KUKA KRL program: EPS_2_251349_MH89A_A_20250929014701.src

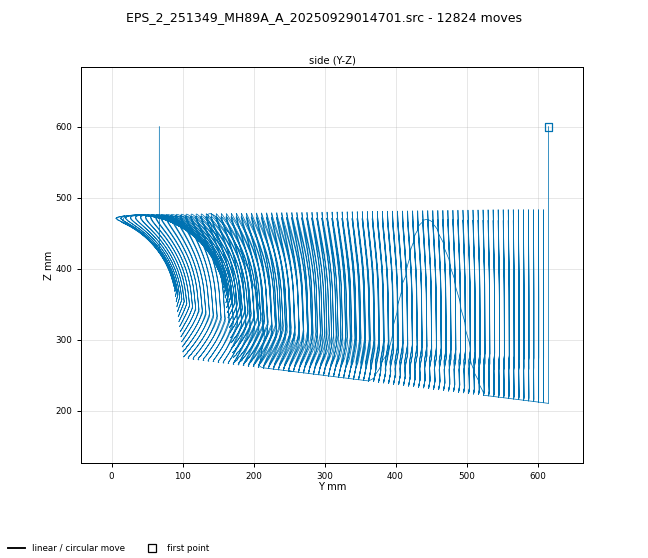
[picture p0: tool path of EPS_2_251349_MH89A_A_20250929014701.src, 12824 of 12826 moves have a stored position in this frame; points joined in program order, loops and branches not executed]
&ACCESS RVP
&REL 4
&COMMENT QRS 19112012
&PARAM EDITMASK = *
DEF PART()
EXT BAS (BAS_COMMAND :IN,REAL :IN )
INT I
BAS (#INITMOV,0 )

;KUKA QRS Post kuka4.cps  Date:22-06-2017 !

File_ID=2864

QRS_PRE_INIT()

;Init var - Until changes are made in qrs_pre_init
Outlet_Square_prg=0
Inlet_1_Square_prg=0
Inlet_2_Square_prg=0
Inlet_3_Square_prg=0
Inlet_4_Square_prg=0
Inlet_5_Square_prg=0

Outlet_1={X 0.000, Y 540.910, Z 382.500, B 0.000, E1 0.000 }
Inlet_1={X 0.000, Y 541.980, Z 367.500, B 0.000, E1 157.000 }
Outlet_1_type=201
Inlet_1_type=201
;QRS#1=Sidecore dimensions
;QRS#2=200-8" PVC SDR 35
;QRS#3=200-8" PVC SDR 35
;QRS#4=
;QRS#5=
;QRS#6=
;QRS#7=
;QRS#8=
;QRS#9=12-08 PSX
;QRS#10=12-08 PSX
;QRS#11=
;QRS#12=
;QRS#13=
;QRS#14=
;QRS#15=
;QRS#16=1220x127x762 2,5'
;QRS#17=EPS Height
;QRS#18=483
;QRS#19=*
;QRS#20= UPDATED VERSION 22-06-2017
;QRS#21=*
Outlet_Square=0100
Inlet_1_Square=0100
Inlet_2_Square=0
Inlet_3_Square=0
Inlet_4_Square=0
Inlet_5_Square=0
Mill_Square=1
Outlet_Square_Prg=204
Inlet_1_Square_prg=204

QRS_INIT()

$ADVANCE=5

; T1
PTP {E1 173.665,E2 173.665}
PTP {X 0,Y 615.418,A -85,B 0,C 180,E1 173.665,E2 173.665,E3 0,E4 0,E5 0,E6 0}
QRS_SPEED_INIT()
LIN {X 0,Y 615.418,Z 600,A -85,B 0,C 180,E1 173.665,E2 173.665,E3 0,E4 0,E5 0,E6 0} C_VEL
LIN {X 0,Y 615.418,Z 220.378,A -85,B 0,C 180,E1 173.665,E2 173.665} C_VEL
LIN {X 0,Y 615.418,Z 212.2,A -85,B 0,C 180,E1 173.665,E2 173.665} C_VEL
LIN {X 0,Y 615.407,Z 210.2,A -85,B 0,C 180,E1 173.479,E2 173.479} C_VEL
LIN {X 0,Y 615.411,Z 210.199,A -85,B 0,C 180,E1 171.465,E2 171.465} C_VEL
LIN {X 0,Y 615.419,Z 210.199,A -85,B 0,C 180,E1 169.475,E2 169.475} C_VEL
LIN {X 0,Y 615.425,Z 210.198,A -85,B 0,C 180,E1 167.471,E2 167.471} C_VEL
LIN {X 0,Y 615.431,Z 210.197,A -85,B 0,C 180,E1 165.452,E2 165.452} C_VEL
LIN {X 0,Y 615.437,Z 210.196,A -85,B 0,C 180,E1 163.415,E2 163.415} C_VEL
LIN {X 0,Y 615.44,Z 210.196,A -85,B 0,C 180,E1 161.356,E2 161.356} C_VEL
LIN {X 0,Y 615.441,Z 210.195,A -85,B 0,C 180,E1 159.271,E2 159.271} C_VEL
LIN {X 0,Y 615.438,Z 210.195,A -85,B 0,C 180,E1 157.157,E2 157.157} C_VEL
LIN {X 0,Y 615.434,Z 210.194,A -85,B 0,C 180,E1 155.009,E2 155.009} C_VEL
LIN {X 0,Y 615.429,Z 210.194,A -85,B 0,C 180,E1 152.824,E2 152.824} C_VEL
LIN {X 0,Y 615.425,Z 210.195,A -85,B 0,C 180,E1 150.594,E2 150.594} C_VEL
LIN {X 0,Y 615.425,Z 210.196,A -85,B 0,C 180,E1 148.315,E2 148.315} C_VEL
LIN {X 0,Y 615.44,Z 210.197,A -85,B 0,C 180,E1 145.979,E2 145.979} C_VEL
LIN {X 0,Y 615.468,Z 210.2,A -85,B 0,C 180,E1 143.578,E2 143.578} C_VEL
LIN {X 0,Y 615.489,Z 210.188,A -85,B 0,C 180,E1 140.936,E2 140.936} C_VEL
LIN {X 0,Y 615.454,Z 210.19,A -85,B 0,C 180,E1 138.528,E2 138.528} C_VEL
LIN {X 0,Y 615.437,Z 210.193,A -85,B 0,C 180,E1 136.006,E2 136.006} C_VEL
LIN {X 0,Y 615.439,Z 210.192,A -85,B 0,C 180,E1 133.998,E2 133.998} C_VEL
LIN {X 0,Y 615.491,Z 210.391,A -85,B 0,C 180,E1 133.031,E2 133.031} C_VEL
LIN {X 0,Y 615.494,Z 227.3,A -85,B 0,C 180,E1 130.35,E2 130.35} C_VEL
LIN {X 0,Y 615.432,Z 244.862,A -85,B 0,C 180,E1 127.63,E2 127.63} C_VEL
LIN {X 0,Y 615.441,Z 256.667,A -85,B 0,C 180,E1 125.853,E2 125.853} C_VEL
LIN {X 0,Y 615.439,Z 257.703,A -85,B 0,C 180,E1 125.807,E2 125.807} C_VEL
LIN {X 0,Y 615.498,Z 364.309,A -85,B 0,C 180,E1 124.535,E2 124.535} C_VEL
LIN {X 0,Y 615.496,Z 377.737,A -85,B 0,C 180,E1 124.235,E2 124.235} C_VEL
LIN {X 0,Y 615.497,Z 389.639,A -85,B 0,C 180,E1 123.841,E2 123.841} C_VEL
LIN {X 0,Y 615.48,Z 401.538,A -85,B 0,C 180,E1 123.313,E2 123.313} C_VEL
LIN {X 0,Y 615.477,Z 412.999,A -85,B 0,C 180,E1 122.651,E2 122.651} C_VEL
LIN {X 0,Y 615.498,Z 424.079,A -85,B 0,C 180,E1 121.847,E2 121.847} C_VEL
LIN {X 0,Y 615.495,Z 432.368,A -85,B 0,C 180,E1 121.095,E2 121.095} C_VEL
LIN {X 0,Y 615.493,Z 439.497,A -85,B 0,C 180,E1 120.348,E2 120.348} C_VEL
LIN {X 0,Y 615.487,Z 446.811,A -85,B 0,C 180,E1 119.405,E2 119.405} C_VEL
LIN {X 0,Y 615.496,Z 452.759,A -85,B 0,C 180,E1 118.46,E2 118.46} C_VEL
LIN {X 0,Y 615.495,Z 457.422,A -85,B 0,C 180,E1 117.544,E2 117.544} C_VEL
LIN {X 0,Y 615.496,Z 461.71,A -85,B 0,C 180,E1 116.443,E2 116.443} C_VEL
LIN {X 0,Y 615.494,Z 464.217,A -85,B 0,C 180,E1 115.579,E2 115.579} C_VEL
LIN {X 0,Y 615.498,Z 465.487,A -85,B 0,C 180,E1 114.99,E2 114.99} C_VEL
LIN {X 0,Y 615.495,Z 466.868,A -85,B 0,C 180,E1 114.02,E2 114.02} C_VEL
LIN {X 0,Y 615.492,Z 467.368,A -85,B 0,C 180,E1 112.844,E2 112.844} C_VEL
LIN {X 0,Y 615.497,Z 467.056,A -85,B 0,C 180,E1 112.135,E2 112.135} C_VEL
LIN {X 0,Y 615.496,Z 466.325,A -85,B 0,C 180,E1 111.431,E2 111.431} C_VEL
LIN {X 0,Y 615.496,Z 464.751,A -85,B 0,C 180,E1 110.571,E2 110.571} C_VEL
LIN {X 0,Y 615.497,Z 461.291,A -85,B 0,C 180,E1 109.337,E2 109.337} C_VEL
LIN {X 0,Y 615.496,Z 457.068,A -85,B 0,C 180,E1 108.287,E2 108.287} C_VEL
LIN {X 0,Y 615.497,Z 450.678,A -85,B 0,C 180,E1 107.098,E2 107.098} C_VEL
LIN {X 0,Y 615.498,Z 443.391,A -85,B 0,C 180,E1 106.04,E2 106.04} C_VEL
LIN {X 0,Y 615.497,Z 436.479,A -85,B 0,C 180,E1 105.225,E2 105.225} C_VEL
LIN {X 0,Y 615.498,Z 426.304,A -85,B 0,C 180,E1 104.251,E2 104.251} C_VEL
LIN {X 0,Y 615.492,Z 415.94,A -85,B 0,C 180,E1 103.453,E2 103.453} C_VEL
LIN {X 0,Y 615.47,Z 405,A -85,B 0,C 180,E1 102.781,E2 102.781} C_VEL
LIN {X 0,Y 615.498,Z 392.743,A -85,B 0,C 180,E1 102.194,E2 102.194} C_VEL
LIN {X 0,Y 615.498,Z 379.878,A -85,B 0,C 180,E1 101.735,E2 101.735} C_VEL
LIN {X 0,Y 615.498,Z 366.871,A -85,B 0,C 180,E1 101.422,E2 101.422} C_VEL
LIN {X 0,Y 615.496,Z 348.647,A -85,B 0,C 180,E1 101.174,E2 101.174} C_VEL
LIN {X 0,Y 615.43,Z 257.274,A -85,B 0,C 180,E1 100.091,E2 100.091} C_VEL
LIN {X 0,Y 615.432,Z 256.35,A -85,B 0,C 180,E1 100.029,E2 100.029} C_VEL
LIN {X 0,Y 615.495,Z 239.011,A -85,B 0,C 180,E1 97.38,E2 97.38} C_VEL
LIN {X 0,Y 615.47,Z 221.075,A -85,B 0,C 180,E1 94.584,E2 94.584} C_VEL
LIN {X 0,Y 615.498,Z 210.337,A -85,B 0,C 180,E1 92.863,E2 92.863} C_VEL
LIN {X 0,Y 615.484,Z 210.201,A -85,B 0,C 180,E1 90.654,E2 90.654} C_VEL
LIN {X 0,Y 615.432,Z 210.196,A -85,B 0,C 180,E1 88.036,E2 88.036} C_VEL
LIN {X 0,Y 615.437,Z 210.197,A -85,B 0,C 180,E1 86.071,E2 86.071} C_VEL
LIN {X 0,Y 615.445,Z 210.198,A -85,B 0,C 180,E1 84.101,E2 84.101} C_VEL
LIN {X 0,Y 615.453,Z 210.198,A -85,B 0,C 180,E1 82.123,E2 82.123} C_VEL
LIN {X 0,Y 615.462,Z 210.199,A -85,B 0,C 180,E1 80.137,E2 80.137} C_VEL
LIN {X 0,Y 615.419,Z 210.197,A -85,B 0,C 180,E1 77.468,E2 77.468} C_VEL
LIN {X 0,Y 615.42,Z 210.197,A -85,B 0,C 180,E1 75.449,E2 75.449} C_VEL
LIN {X 0,Y 615.419,Z 210.197,A -85,B 0,C 180,E1 73.411,E2 73.411} C_VEL
LIN {X 0,Y 615.419,Z 210.197,A -85,B 0,C 180,E1 71.351,E2 71.351} C_VEL
LIN {X 0,Y 615.417,Z 210.198,A -85,B 0,C 180,E1 69.266,E2 69.266} C_VEL
LIN {X 0,Y 615.415,Z 210.198,A -85,B 0,C 180,E1 67.152,E2 67.152} C_VEL
LIN {X 0,Y 615.412,Z 210.198,A -85,B 0,C 180,E1 65.005,E2 65.005} C_VEL
LIN {X 0,Y 615.411,Z 210.198,A -85,B 0,C 180,E1 62.819,E2 62.819} C_VEL
LIN {X 0,Y 615.444,Z 210.197,A -85,B 0,C 180,E1 60.205,E2 60.205} C_VEL
LIN {X 0,Y 615.478,Z 210.2,A -85,B 0,C 180,E1 57.542,E2 57.542} C_VEL
LIN {X 0,Y 615.438,Z 210.2,A -85,B 0,C 180,E1 55.181,E2 55.181} C_VEL
LIN {X 0,Y 615.409,Z 210.199,A -85,B 0,C 180,E1 52.752,E2 52.752} C_VEL
LIN {X 0,Y 615.406,Z 210.2,A -85,B 0,C 180,E1 50.243,E2 50.243} C_VEL
LIN {X 0,Y 615.451,Z 210.2,A -85,B 0,C 180,E1 47.644,E2 47.644} C_VEL
LIN {X 0,Y 615.447,Z 210.2,A -85,B 0,C 180,E1 44.927,E2 44.927} C_VEL
LIN {X 0,Y 615.471,Z 210.2,A -85,B 0,C 180,E1 43.045,E2 43.045} C_VEL
LIN {X 0,Y 615.43,Z 210.199,A -85,B 0,C 180,E1 40.606,E2 40.606} C_VEL
LIN {X 0,Y 615.48,Z 210.198,A -85,B 0,C 180,E1 38.9,E2 38.9} C_VEL
LIN {X 0,Y 615.43,Z 210.198,A -85,B 0,C 180,E1 36.425,E2 36.425} C_VEL
LIN {X 0,Y 615.411,Z 210.198,A -85,B 0,C 180,E1 34.023,E2 34.023} C_VEL
LIN {X 0,Y 615.411,Z 210.198,A -85,B 0,C 180,E1 31.686,E2 31.686} C_VEL
LIN {X 0,Y 615.42,Z 210.198,A -85,B 0,C 180,E1 29.406,E2 29.406} C_VEL
LIN {X 0,Y 615.447,Z 210.199,A -85,B 0,C 180,E1 27.037,E2 27.037} C_VEL
LIN {X 0,Y 615.439,Z 210.195,A -85,B 0,C 180,E1 23.998,E2 23.998} C_VEL
LIN {X 0,Y 615.463,Z 210.194,A -85,B 0,C 180,E1 22.134,E2 22.134} C_VEL
LIN {X 0,Y 615.461,Z 210.194,A -85,B 0,C 180,E1 20.031,E2 20.031} C_VEL
LIN {X 0,Y 615.462,Z 210.193,A -85,B 0,C 180,E1 17.955,E2 17.955} C_VEL
LIN {X 0,Y 615.466,Z 210.193,A -85,B 0,C 180,E1 15.903,E2 15.903} C_VEL
LIN {X 0,Y 615.422,Z 210.195,A -85,B 0,C 180,E1 13.2,E2 13.2} C_VEL
LIN {X 0,Y 615.424,Z 210.197,A -85,B 0,C 180,E1 10.857,E2 10.857} C_VEL
LIN {X 0,Y 615.442,Z 210.198,A -85,B 0,C 180,E1 8.535,E2 8.535} C_VEL
LIN {X 0,Y 615.497,Z 210.196,A -85,B 0,C 180,E1 5.896,E2 5.896} C_VEL
LIN {X 0,Y 615.452,Z 210.191,A -85,B 0,C 180,E1 3.271,E2 3.271} C_VEL
LIN {X 0,Y 615.465,Z 210.19,A -85,B 0,C 180,E1 1.306,E2 1.306} C_VEL
LIN {X 0,Y 615.43,Z 210.194,A -85,B 0,C 180,E1 -1.311,E2 -1.311} C_VEL
LIN {X 0,Y 615.434,Z 210.192,A -85,B 0,C 180,E1 -3.275,E2 -3.275} C_VEL
LIN {X 0,Y 615.439,Z 210.192,A -85,B 0,C 180,E1 -5.244,E2 -5.244} C_VEL
LIN {X 0,Y 615.448,Z 210.19,A -85,B 0,C 180,E1 -7.218,E2 -7.218} C_VEL
LIN {X 0,Y 615.456,Z 210.189,A -85,B 0,C 180,E1 -9.201,E2 -9.201} C_VEL
LIN {X 0,Y 615.465,Z 210.188,A -85,B 0,C 180,E1 -11.195,E2 -11.195} C_VEL
LIN {X 0,Y 615.472,Z 210.188,A -85,B 0,C 180,E1 -13.203,E2 -13.203} C_VEL
LIN {X 0,Y 615.438,Z 210.193,A -85,B 0,C 180,E1 -15.908,E2 -15.908} C_VEL
LIN {X 0,Y 615.473,Z 210.199,A -85,B 0,C 180,E1 -18.6,E2 -18.6} C_VEL
LIN {X 0,Y 615.484,Z 210.185,A -85,B 0,C 180,E1 -21.434,E2 -21.434} C_VEL
LIN {X 0,Y 615.445,Z 210.19,A -85,B 0,C 180,E1 -23.999,E2 -23.999} C_VEL
LIN {X 0,Y 615.444,Z 210.194,A -85,B 0,C 180,E1 -26.448,E2 -26.448} C_VEL
LIN {X 0,Y 615.493,Z 210.191,A -85,B 0,C 180,E1 -29.407,E2 -29.407} C_VEL
LIN {X 0,Y 615.489,Z 210.186,A -85,B 0,C 180,E1 -31.687,E2 -31.687} C_VEL
LIN {X 0,Y 615.473,Z 210.185,A -85,B 0,C 180,E1 -34.024,E2 -34.024} C_VEL
LIN {X 0,Y 615.451,Z 210.189,A -85,B 0,C 180,E1 -36.429,E2 -36.429} C_VEL
LIN {X 0,Y 615.46,Z 210.195,A -85,B 0,C 180,E1 -39.059,E2 -39.059} C_VEL
LIN {X 0,Y 615.49,Z 210.201,A -85,B 0,C 180,E1 -41.475,E2 -41.475} C_VEL
LIN {X 0,Y 615.496,Z 210.183,A -85,B 0,C 180,E1 -44.15,E2 -44.15} C_VEL
LIN {X 0,Y 615.453,Z 210.19,A -85,B 0,C 180,E1 -46.957,E2 -46.957} C_VEL
LIN {X 0,Y 615.463,Z 210.195,A -85,B 0,C 180,E1 -49.391,E2 -49.391} C_VEL
LIN {X 0,Y 615.493,Z 210.196,A -85,B 0,C 180,E1 -51.989,E2 -51.989} C_VEL
LIN {X 0,Y 615.49,Z 210.187,A -85,B 0,C 180,E1 -54.384,E2 -54.384} C_VEL
LIN {X 0,Y 615.486,Z 210.182,A -85,B 0,C 180,E1 -56.763,E2 -56.763} C_VEL
LIN {X 0,Y 615.472,Z 210.184,A -85,B 0,C 180,E1 -59.079,E2 -59.079} C_VEL
LIN {X 0,Y 615.46,Z 210.19,A -85,B 0,C 180,E1 -61.556,E2 -61.556} C_VEL
LIN {X 0,Y 615.498,Z 210.199,A -85,B 0,C 180,E1 -64.284,E2 -64.284} C_VEL
LIN {X 0,Y 615.484,Z 210.182,A -85,B 0,C 180,E1 -67.155,E2 -67.155} C_VEL
LIN {X 0,Y 615.492,Z 210.437,A -85,B 0,C 180,E1 -68.48,E2 -68.48} C_VEL
LIN {X 0,Y 615.494,Z 228.957,A -85,B 0,C 180,E1 -71.181,E2 -71.181} C_VEL
LIN {X 0,Y 615.488,Z 249.421,A -85,B 0,C 180,E1 -74.094,E2 -74.094} C_VEL
LIN {X 0,Y 615.473,Z 268.661,A -85,B 0,C 180,E1 -76.798,E2 -76.798} C_VEL
LIN {X 0,Y 615.487,Z 271.24,A -85,B 0,C 180,E1 -77.113,E2 -77.113} C_VEL
LIN {X 0,Y 615.491,Z 280.005,A -85,B 0,C 180,E1 -77.239,E2 -77.239} C_VEL
LIN {X 0,Y 615.498,Z 378.802,A -85,B 0,C 180,E1 -78.41,E2 -78.41} C_VEL
LIN {X 0,Y 615.498,Z 391.325,A -85,B 0,C 180,E1 -78.682,E2 -78.682} C_VEL
LIN {X 0,Y 615.496,Z 404.513,A -85,B 0,C 180,E1 -79.109,E2 -79.109} C_VEL
LIN {X 0,Y 615.491,Z 416.467,A -85,B 0,C 180,E1 -79.639,E2 -79.639} C_VEL
LIN {X 0,Y 615.48,Z 427.989,A -85,B 0,C 180,E1 -80.303,E2 -80.303} C_VEL
LIN {X 0,Y 615.499,Z 438.335,A -85,B 0,C 180,E1 -81.049,E2 -81.049} C_VEL
LIN {X 0,Y 615.498,Z 446.687,A -85,B 0,C 180,E1 -81.794,E2 -81.794} C_VEL
LIN {X 0,Y 615.498,Z 454.602,A -85,B 0,C 180,E1 -82.619,E2 -82.619} C_VEL
LIN {X 0,Y 615.49,Z 462.201,A -85,B 0,C 180,E1 -83.607,E2 -83.607} C_VEL
LIN {X 0,Y 615.498,Z 469.202,A -85,B 0,C 180,E1 -84.758,E2 -84.758} C_VEL
LIN {X 0,Y 615.493,Z 473.849,A -85,B 0,C 180,E1 -85.743,E2 -85.743} C_VEL
LIN {X 0,Y 615.494,Z 477.397,A -85,B 0,C 180,E1 -86.727,E2 -86.727} C_VEL
LIN {X 0,Y 615.497,Z 479.232,A -85,B 0,C 180,E1 -87.382,E2 -87.382} C_VEL
LIN {X 0,Y 615.497,Z 480.607,A -85,B 0,C 180,E1 -88.036,E2 -88.036} C_VEL
LIN {X 0,Y 615.496,Z 482.173,A -85,B 0,C 180,E1 -89.345,E2 -89.345} C_VEL
LIN {X 0,Y 615.494,Z 482.389,A -85,B 0,C 180,E1 -89.999,E2 -89.999} C_VEL
LIN {X 0,Y 615.495,Z 481.581,A -85,B 0,C 180,E1 -91.308,E2 -91.308} C_VEL
LIN {X 0,Y 615.497,Z 480.609,A -85,B 0,C 180,E1 -91.963,E2 -91.963} C_VEL
LIN {X 0,Y 615.497,Z 479.234,A -85,B 0,C 180,E1 -92.617,E2 -92.617} C_VEL
LIN {X 0,Y 615.496,Z 476.351,A -85,B 0,C 180,E1 -93.6,E2 -93.6} C_VEL
LIN {X 0,Y 615.498,Z 472.444,A -85,B 0,C 180,E1 -94.584,E2 -94.584} C_VEL
LIN {X 0,Y 615.499,Z 467.408,A -85,B 0,C 180,E1 -95.569,E2 -95.569} C_VEL
LIN {X 0,Y 615.489,Z 460.918,A -85,B 0,C 180,E1 -96.577,E2 -96.577} C_VEL
LIN {X 0,Y 615.497,Z 453.138,A -85,B 0,C 180,E1 -97.545,E2 -97.545} C_VEL
LIN {X 0,Y 615.498,Z 443.264,A -85,B 0,C 180,E1 -98.536,E2 -98.536} C_VEL
LIN {X 0,Y 615.495,Z 432.874,A -85,B 0,C 180,E1 -99.364,E2 -99.364} C_VEL
LIN {X 0,Y 615.475,Z 422.588,A -85,B 0,C 180,E1 -100.028,E2 -100.028} C_VEL
LIN {X 0,Y 615.497,Z 411.108,A -85,B 0,C 180,E1 -100.617,E2 -100.617} C_VEL
LIN {X 0,Y 615.499,Z 399.282,A -85,B 0,C 180,E1 -101.079,E2 -101.079} C_VEL
LIN {X 0,Y 615.498,Z 386.267,A -85,B 0,C 180,E1 -101.442,E2 -101.442} C_VEL
LIN {X 0,Y 615.499,Z 372.989,A -85,B 0,C 180,E1 -101.672,E2 -101.672} C_VEL
LIN {X 0,Y 615.488,Z 271.757,A -85,B 0,C 180,E1 -102.865,E2 -102.865} C_VEL
LIN {X 0,Y 615.485,Z 270.524,A -85,B 0,C 180,E1 -102.949,E2 -102.949} C_VEL
LIN {X 0,Y 615.481,Z 250.632,A -85,B 0,C 180,E1 -105.735,E2 -105.735} C_VEL
LIN {X 0,Y 615.491,Z 231.586,A -85,B 0,C 180,E1 -108.442,E2 -108.442} C_VEL
LIN {X 0,Y 615.492,Z 212.096,A -85,B 0,C 180,E1 -111.255,E2 -111.255} C_VEL
LIN {X 0,Y 615.49,Z 210.315,A -85,B 0,C 180,E1 -111.563,E2 -111.563} C_VEL
LIN {X 0,Y 615.461,Z 210.19,A -85,B 0,C 180,E1 -114.272,E2 -114.272} C_VEL
LIN {X 0,Y 615.497,Z 210.18,A -85,B 0,C 180,E1 -117.046,E2 -117.046} C_VEL
LIN {X 0,Y 615.497,Z 210.199,A -85,B 0,C 180,E1 -119.795,E2 -119.795} C_VEL
LIN {X 0,Y 615.457,Z 210.192,A -85,B 0,C 180,E1 -122.458,E2 -122.458} C_VEL
LIN {X 0,Y 615.456,Z 210.188,A -85,B 0,C 180,E1 -124.816,E2 -124.816} C_VEL
LIN {X 0,Y 615.476,Z 210.184,A -85,B 0,C 180,E1 -127.242,E2 -127.242} C_VEL
LIN {X 0,Y 615.497,Z 210.199,A -85,B 0,C 180,E1 -130.089,E2 -130.089} C_VEL
LIN {X 0,Y 615.481,Z 210.198,A -85,B 0,C 180,E1 -132.352,E2 -132.352} C_VEL
LIN {X 0,Y 615.444,Z 210.191,A -85,B 0,C 180,E1 -135.071,E2 -135.071} C_VEL
LIN {X 0,Y 615.498,Z 210.185,A -85,B 0,C 180,E1 -137.917,E2 -137.917} C_VEL
LIN {X 0,Y 615.495,Z 210.194,A -85,B 0,C 180,E1 -140.249,E2 -140.249} C_VEL
LIN {X 0,Y 615.445,Z 210.195,A -85,B 0,C 180,E1 -143.067,E2 -143.067} C_VEL
LIN {X 0,Y 615.438,Z 210.193,A -85,B 0,C 180,E1 -145.304,E2 -145.304} C_VEL
LIN {X 0,Y 615.441,Z 210.191,A -85,B 0,C 180,E1 -147.674,E2 -147.674} C_VEL
LIN {X 0,Y 615.491,Z 210.197,A -85,B 0,C 180,E1 -150.592,E2 -150.592} C_VEL
LIN {X 0,Y 615.476,Z 210.199,A -85,B 0,C 180,E1 -152.955,E2 -152.955} C_VEL
LIN {X 0,Y 615.476,Z 210.199,A -85,B 0,C 180,E1 -155.006,E2 -155.006} C_VEL
LIN {X 0,Y 615.429,Z 210.195,A -85,B 0,C 180,E1 -157.665,E2 -157.665} C_VEL
LIN {X 0,Y 615.424,Z 210.195,A -85,B 0,C 180,E1 -159.963,E2 -159.963} C_VEL
LIN {X 0,Y 615.481,Z 210.192,A -85,B 0,C 180,E1 -162.728,E2 -162.728} C_VEL
LIN {X 0,Y 615.455,Z 210.199,A -85,B 0,C 180,E1 -165.448,E2 -165.448} C_VEL
LIN {X 0,Y 615.46,Z 210.199,A -85,B 0,C 180,E1 -167.467,E2 -167.467} C_VEL
LIN {X 0,Y 615.463,Z 210.2,A -85,B 0,C 180,E1 -169.471,E2 -169.471} C_VEL
LIN {X 0,Y 615.416,Z 210.198,A -85,B 0,C 180,E1 -172.121,E2 -172.121} C_VEL
LIN {X 0,Y 615.417,Z 210.198,A -85,B 0,C 180,E1 -174.099,E2 -174.099} C_VEL
LIN {X 0,Y 615.419,Z 210.199,A -85,B 0,C 180,E1 -176.069,E2 -176.069} C_VEL
LIN {X 0,Y 615.427,Z 210.199,A -85,B 0,C 180,E1 -178.035,E2 -178.035} C_VEL
LIN {X 0,Y 615.434,Z 210.2,A -85,B 0,C 180,E1 -179.998,E2 -179.998} C_VEL
LIN {X 0,Y 615.444,Z 210.2,A -85,B 0,C 180,E1 -181.961,E2 -181.961} C_VEL
LIN {X 0,Y 615.403,Z 210.2,A -85,B 0,C 180,E1 -184.583,E2 -184.583} C_VEL
LIN {X 0,Y 615.407,Z 210.2,A -85,B 0,C 180,E1 -186.521,E2 -186.521} C_VEL
LIN {X 0,Y 614.735,Z 210.347,A -85,B 0,C 180,E1 -187.068,E2 -187.068} C_VEL
LIN {X 0,Y 611.898,Z 210.766,A -85,B 0,C 180,E1 -187.954,E2 -187.954} C_VEL
LIN {X 0,Y 609.512,Z 211.071,A -85,B 0,C 180,E1 -188.667,E2 -188.667} C_VEL
LIN {X 0,Y 608.496,Z 211.185,A -85,B 0,C 180,E1 -189.217,E2 -189.217} C_VEL
LIN {X 0,Y 608.417,Z 211.194,A -85,B 0,C 180,E1 -189.403,E2 -189.403} C_VEL
LIN {X 0,Y 608.444,Z 211.197,A -85,B 0,C 180,E1 -191.997,E2 -191.997} C_VEL
LIN {X 0,Y 608.389,Z 211.195,A -85,B 0,C 180,E1 -194.72,E2 -194.72} C_VEL
LIN {X 0,Y 608.4,Z 211.193,A -85,B 0,C 180,E1 -196.783,E2 -196.783} C_VEL
LIN {X 0,Y 608.415,Z 211.192,A -85,B 0,C 180,E1 -198.868,E2 -198.868} C_VEL
LIN {X 0,Y 608.41,Z 211.192,A -85,B 0,C 180,E1 -200.98,E2 -200.98} C_VEL
LIN {X 0,Y 608.401,Z 211.193,A -85,B 0,C 180,E1 -203.123,E2 -203.123} C_VEL
LIN {X 0,Y 608.392,Z 211.194,A -85,B 0,C 180,E1 -205.3,E2 -205.3} C_VEL
LIN {X 0,Y 608.404,Z 211.193,A -85,B 0,C 180,E1 -207.517,E2 -207.517} C_VEL
LIN {X 0,Y 608.424,Z 211.194,A -85,B 0,C 180,E1 -209.966,E2 -209.966} C_VEL
LIN {X 0,Y 608.435,Z 211.193,A -85,B 0,C 180,E1 -212.877,E2 -212.877} C_VEL
LIN {X 0,Y 608.415,Z 211.192,A -85,B 0,C 180,E1 -215.275,E2 -215.275} C_VEL
LIN {X 0,Y 608.428,Z 211.189,A -85,B 0,C 180,E1 -217.745,E2 -217.745} C_VEL
LIN {X 0,Y 608.42,Z 211.195,A -85,B 0,C 180,E1 -220.327,E2 -220.327} C_VEL
LIN {X 0,Y 608.473,Z 211.187,A -85,B 0,C 180,E1 -223.31,E2 -223.31} C_VEL
LIN {X 0,Y 608.43,Z 211.191,A -85,B 0,C 180,E1 -226.128,E2 -226.128} C_VEL
LIN {X 0,Y 608.49,Z 211.355,A -85,B 0,C 180,E1 -226.881,E2 -226.881} C_VEL
LIN {X 0,Y 608.513,Z 227.639,A -85,B 0,C 180,E1 -229.486,E2 -229.486} C_VEL
LIN {X 0,Y 608.436,Z 245.336,A -85,B 0,C 180,E1 -232.252,E2 -232.252} C_VEL
LIN {X 0,Y 608.443,Z 256.928,A -85,B 0,C 180,E1 -234.011,E2 -234.011} C_VEL
LIN {X 0,Y 608.525,Z 261.477,A -85,B 0,C 180,E1 -234.093,E2 -234.093} C_VEL
LIN {X 0,Y 608.569,Z 363.854,A -85,B 0,C 180,E1 -235.32,E2 -235.32} C_VEL
LIN {X 0,Y 608.535,Z 376.972,A -85,B 0,C 180,E1 -235.61,E2 -235.61} C_VEL
LIN {X 0,Y 608.533,Z 389.666,A -85,B 0,C 180,E1 -236.029,E2 -236.029} C_VEL
LIN {X 0,Y 608.501,Z 400.985,A -85,B 0,C 180,E1 -236.531,E2 -236.531} C_VEL
LIN {X 0,Y 608.474,Z 411.466,A -85,B 0,C 180,E1 -237.122,E2 -237.122} C_VEL
LIN {X 0,Y 608.482,Z 422.54,A -85,B 0,C 180,E1 -237.907,E2 -237.907} C_VEL
LIN {X 0,Y 608.461,Z 431.398,A -85,B 0,C 180,E1 -238.684,E2 -238.684} C_VEL
LIN {X 0,Y 608.47,Z 440.256,A -85,B 0,C 180,E1 -239.614,E2 -239.614} C_VEL
LIN {X 0,Y 608.45,Z 447.768,A -85,B 0,C 180,E1 -240.601,E2 -240.601} C_VEL
LIN {X 0,Y 608.443,Z 454.63,A -85,B 0,C 180,E1 -241.734,E2 -241.734} C_VEL
LIN {X 0,Y 608.431,Z 459.601,A -85,B 0,C 180,E1 -242.793,E2 -242.793} C_VEL
LIN {X 0,Y 608.427,Z 463.656,A -85,B 0,C 180,E1 -243.964,E2 -243.964} C_VEL
LIN {X 0,Y 608.436,Z 465.478,A -85,B 0,C 180,E1 -244.699,E2 -244.699} C_VEL
LIN {X 0,Y 608.422,Z 467.335,A -85,B 0,C 180,E1 -245.85,E2 -245.85} C_VEL
LIN {X 0,Y 608.427,Z 467.966,A -85,B 0,C 180,E1 -246.876,E2 -246.876} C_VEL
LIN {X 0,Y 608.428,Z 467.862,A -85,B 0,C 180,E1 -247.594,E2 -247.594} C_VEL
LIN {X 0,Y 608.416,Z 467.256,A -85,B 0,C 180,E1 -248.307,E2 -248.307} C_VEL
LIN {X 0,Y 608.433,Z 465.634,A -85,B 0,C 180,E1 -249.319,E2 -249.319} C_VEL
LIN {X 0,Y 608.424,Z 462.722,A -85,B 0,C 180,E1 -250.429,E2 -250.429} C_VEL
LIN {X 0,Y 608.441,Z 458.5,A -85,B 0,C 180,E1 -251.554,E2 -251.554} C_VEL
LIN {X 0,Y 608.435,Z 453.717,A -85,B 0,C 180,E1 -252.524,E2 -252.524} C_VEL
LIN {X 0,Y 608.438,Z 447.923,A -85,B 0,C 180,E1 -253.466,E2 -253.466} C_VEL
LIN {X 0,Y 608.469,Z 440.69,A -85,B 0,C 180,E1 -254.423,E2 -254.423} C_VEL
LIN {X 0,Y 608.485,Z 432.669,A -85,B 0,C 180,E1 -255.28,E2 -255.28} C_VEL
LIN {X 0,Y 608.476,Z 425.263,A -85,B 0,C 180,E1 -255.963,E2 -255.963} C_VEL
LIN {X 0,Y 608.483,Z 415.088,A -85,B 0,C 180,E1 -256.73,E2 -256.73} C_VEL
LIN {X 0,Y 608.488,Z 403.825,A -85,B 0,C 180,E1 -257.409,E2 -257.409} C_VEL
LIN {X 0,Y 608.535,Z 391.188,A -85,B 0,C 180,E1 -258.002,E2 -258.002} C_VEL
LIN {X 0,Y 608.539,Z 378.189,A -85,B 0,C 180,E1 -258.446,E2 -258.446} C_VEL
LIN {X 0,Y 608.549,Z 365.289,A -85,B 0,C 180,E1 -258.743,E2 -258.743} C_VEL
LIN {X 0,Y 608.548,Z 330.21,A -85,B 0,C 180,E1 -259.182,E2 -259.182} C_VEL
LIN {X 0,Y 608.449,Z 257.153,A -85,B 0,C 180,E1 -260.065,E2 -260.065} C_VEL
LIN {X 0,Y 608.436,Z 254.884,A -85,B 0,C 180,E1 -260.359,E2 -260.359} C_VEL
LIN {X 0,Y 608.467,Z 236.476,A -85,B 0,C 180,E1 -263.218,E2 -263.218} C_VEL
LIN {X 0,Y 608.521,Z 218.644,A -85,B 0,C 180,E1 -266.027,E2 -266.027} C_VEL
LIN {X 0,Y 608.487,Z 211.297,A -85,B 0,C 180,E1 -267.228,E2 -267.228} C_VEL
LIN {X 0,Y 608.418,Z 211.192,A -85,B 0,C 180,E1 -270.001,E2 -270.001} C_VEL
LIN {X 0,Y 608.402,Z 211.194,A -85,B 0,C 180,E1 -271.986,E2 -271.986} C_VEL
LIN {X 0,Y 608.406,Z 211.194,A -85,B 0,C 180,E1 -273.975,E2 -273.975} C_VEL
LIN {X 0,Y 608.416,Z 211.194,A -85,B 0,C 180,E1 -275.968,E2 -275.968} C_VEL
LIN {X 0,Y 608.439,Z 211.192,A -85,B 0,C 180,E1 -277.968,E2 -277.968} C_VEL
LIN {X 0,Y 608.405,Z 211.192,A -85,B 0,C 180,E1 -280.651,E2 -280.651} C_VEL
LIN {X 0,Y 608.435,Z 211.193,A -85,B 0,C 180,E1 -283.358,E2 -283.358} C_VEL
LIN {X 0,Y 608.431,Z 211.195,A -85,B 0,C 180,E1 -286.095,E2 -286.095} C_VEL
LIN {X 0,Y 608.404,Z 211.192,A -85,B 0,C 180,E1 -288.872,E2 -288.872} C_VEL
LIN {X 0,Y 608.438,Z 211.194,A -85,B 0,C 180,E1 -291.693,E2 -291.693} C_VEL
LIN {X 0,Y 608.41,Z 211.195,A -85,B 0,C 180,E1 -294.573,E2 -294.573} C_VEL
LIN {X 0,Y 608.391,Z 211.194,A -85,B 0,C 180,E1 -297.2,E2 -297.2} C_VEL
LIN {X 0,Y 608.463,Z 211.191,A -85,B 0,C 180,E1 -299.979,E2 -299.979} C_VEL
LIN {X 0,Y 608.412,Z 211.194,A -85,B 0,C 180,E1 -302.883,E2 -302.883} C_VEL
LIN {X 0,Y 608.382,Z 211.195,A -85,B 0,C 180,E1 -305.282,E2 -305.282} C_VEL
LIN {X 0,Y 608.422,Z 211.196,A -85,B 0,C 180,E1 -308.241,E2 -308.241} C_VEL
LIN {X 0,Y 608.391,Z 211.196,A -85,B 0,C 180,E1 -311.182,E2 -311.182} C_VEL
LIN {X 0,Y 608.401,Z 211.193,A -85,B 0,C 180,E1 -313.876,E2 -313.876} C_VEL
LIN {X 0,Y 608.474,Z 211.193,A -85,B 0,C 180,E1 -316.691,E2 -316.691} C_VEL
LIN {X 0,Y 608.438,Z 211.199,A -85,B 0,C 180,E1 -318.827,E2 -318.827} C_VEL
LIN {X 0,Y 608.406,Z 211.192,A -85,B 0,C 180,E1 -321.767,E2 -321.767} C_VEL
LIN {X 0,Y 608.405,Z 211.192,A -85,B 0,C 180,E1 -323.96,E2 -323.96} C_VEL
LIN {X 0,Y 608.391,Z 211.194,A -85,B 0,C 180,E1 -326.329,E2 -326.329} C_VEL
LIN {X 0,Y 608.422,Z 211.194,A -85,B 0,C 180,E1 -328.737,E2 -328.737} C_VEL
LIN {X 0,Y 608.418,Z 211.194,A -85,B 0,C 180,E1 -331.735,E2 -331.735} C_VEL
LIN {X 0,Y 608.412,Z 211.191,A -85,B 0,C 180,E1 -334.291,E2 -334.291} C_VEL
LIN {X 0,Y 608.407,Z 211.194,A -85,B 0,C 180,E1 -336.878,E2 -336.878} C_VEL
LIN {X 0,Y 608.45,Z 211.194,A -85,B 0,C 180,E1 -339.729,E2 -339.729} C_VEL
LIN {X 0,Y 608.403,Z 211.192,A -85,B 0,C 180,E1 -342.525,E2 -342.525} C_VEL
LIN {X 0,Y 608.422,Z 211.19,A -85,B 0,C 180,E1 -344.596,E2 -344.596} C_VEL
LIN {X 0,Y 608.415,Z 211.191,A -85,B 0,C 180,E1 -346.645,E2 -346.645} C_VEL
LIN {X 0,Y 608.393,Z 211.194,A -85,B 0,C 180,E1 -349.082,E2 -349.082} C_VEL
LIN {X 0,Y 608.415,Z 211.193,A -85,B 0,C 180,E1 -351.366,E2 -351.366} C_VEL
LIN {X 0,Y 608.464,Z 211.196,A -85,B 0,C 180,E1 -354.036,E2 -354.036} C_VEL
LIN {X 0,Y 608.423,Z 211.192,A -85,B 0,C 180,E1 -356.691,E2 -356.691} C_VEL
LIN {X 0,Y 608.451,Z 211.189,A -85,B 0,C 180,E1 -358.679,E2 -358.679} C_VEL
LIN {X 0,Y 608.42,Z 211.19,A -85,B 0,C 180,E1 -361.326,E2 -361.326} C_VEL
LIN {X 0,Y 608.405,Z 211.192,A -85,B 0,C 180,E1 -363.313,E2 -363.313} C_VEL
LIN {X 0,Y 608.422,Z 211.19,A -85,B 0,C 180,E1 -365.304,E2 -365.304} C_VEL
LIN {X 0,Y 608.421,Z 211.19,A -85,B 0,C 180,E1 -367.302,E2 -367.302} C_VEL
LIN {X 0,Y 608.44,Z 211.188,A -85,B 0,C 180,E1 -369.308,E2 -369.308} C_VEL
LIN {X 0,Y 608.429,Z 211.19,A -85,B 0,C 180,E1 -371.327,E2 -371.327} C_VEL
LIN {X 0,Y 608.443,Z 211.188,A -85,B 0,C 180,E1 -373.359,E2 -373.359} C_VEL
LIN {X 0,Y 608.455,Z 211.186,A -85,B 0,C 180,E1 -375.408,E2 -375.408} C_VEL
LIN {X 0,Y 608.414,Z 211.193,A -85,B 0,C 180,E1 -378.175,E2 -378.175} C_VEL
LIN {X 0,Y 608.456,Z 211.195,A -85,B 0,C 180,E1 -380.983,E2 -380.983} C_VEL
LIN {X 0,Y 608.439,Z 211.188,A -85,B 0,C 180,E1 -383.848,E2 -383.848} C_VEL
LIN {X 0,Y 608.423,Z 211.19,A -85,B 0,C 180,E1 -386.038,E2 -386.038} C_VEL
LIN {X 0,Y 608.416,Z 211.191,A -85,B 0,C 180,E1 -388.27,E2 -388.27} C_VEL
LIN {X 0,Y 608.428,Z 211.191,A -85,B 0,C 180,E1 -390.549,E2 -390.549} C_VEL
LIN {X 0,Y 608.444,Z 211.192,A -85,B 0,C 180,E1 -392.882,E2 -392.882} C_VEL
LIN {X 0,Y 608.436,Z 211.2,A -85,B 0,C 180,E1 -395.28,E2 -395.28} C_VEL
LIN {X 0,Y 608.461,Z 211.186,A -85,B 0,C 180,E1 -398.239,E2 -398.239} C_VEL
LIN {X 0,Y 608.435,Z 211.194,A -85,B 0,C 180,E1 -401.18,E2 -401.18} C_VEL
LIN {X 0,Y 608.473,Z 211.19,A -85,B 0,C 180,E1 -403.87,E2 -403.87} C_VEL
LIN {X 0,Y 608.452,Z 211.186,A -85,B 0,C 180,E1 -406.694,E2 -406.694} C_VEL
LIN {X 0,Y 608.432,Z 211.189,A -85,B 0,C 180,E1 -408.821,E2 -408.821} C_VEL
LIN {X 0,Y 608.471,Z 211.194,A -85,B 0,C 180,E1 -411.76,E2 -411.76} C_VEL
LIN {X 0,Y 608.436,Z 211.189,A -85,B 0,C 180,E1 -414.722,E2 -414.722} C_VEL
LIN {X 0,Y 608.448,Z 211.187,A -85,B 0,C 180,E1 -417.12,E2 -417.12} C_VEL
LIN {X 0,Y 608.452,Z 211.197,A -85,B 0,C 180,E1 -420.032,E2 -420.032} C_VEL
LIN {X 0,Y 608.487,Z 211.184,A -85,B 0,C 180,E1 -422.792,E2 -422.792} C_VEL
LIN {X 0,Y 608.445,Z 211.188,A -85,B 0,C 180,E1 -425.428,E2 -425.428} C_VEL
LIN {X 0,Y 608.478,Z 211.292,A -85,B 0,C 180,E1 -428.331,E2 -428.331} C_VEL
LIN {X 0,Y 608.551,Z 215.715,A -85,B 0,C 180,E1 -429.022,E2 -429.022} C_VEL
LIN {X 0,Y 608.504,Z 235.021,A -85,B 0,C 180,E1 -431.829,E2 -431.829} C_VEL
LIN {X 0,Y 608.468,Z 254.327,A -85,B 0,C 180,E1 -434.594,E2 -434.594} C_VEL
LIN {X 0,Y 608.497,Z 271.285,A -85,B 0,C 180,E1 -436.962,E2 -436.962} C_VEL
LIN {X 0,Y 608.588,Z 276.47,A -85,B 0,C 180,E1 -437.049,E2 -437.049} C_VEL
LIN {X 0,Y 608.549,Z 378.922,A -85,B 0,C 180,E1 -438.276,E2 -438.276} C_VEL
LIN {X 0,Y 608.548,Z 392.2,A -85,B 0,C 180,E1 -438.572,E2 -438.572} C_VEL
LIN {X 0,Y 608.545,Z 405.337,A -85,B 0,C 180,E1 -439.009,E2 -439.009} C_VEL
LIN {X 0,Y 608.516,Z 416.626,A -85,B 0,C 180,E1 -439.519,E2 -439.519} C_VEL
LIN {X 0,Y 608.468,Z 428.19,A -85,B 0,C 180,E1 -440.19,E2 -440.19} C_VEL
LIN {X 0,Y 608.485,Z 438.588,A -85,B 0,C 180,E1 -440.945,E2 -440.945} C_VEL
LIN {X 0,Y 608.459,Z 446.998,A -85,B 0,C 180,E1 -441.698,E2 -441.698} C_VEL
LIN {X 0,Y 608.471,Z 454.956,A -85,B 0,C 180,E1 -442.533,E2 -442.533} C_VEL
LIN {X 0,Y 608.437,Z 462.3,A -85,B 0,C 180,E1 -443.486,E2 -443.486} C_VEL
LIN {X 0,Y 608.45,Z 467.863,A -85,B 0,C 180,E1 -444.365,E2 -444.365} C_VEL
LIN {X 0,Y 608.432,Z 472.948,A -85,B 0,C 180,E1 -445.362,E2 -445.362} C_VEL
LIN {X 0,Y 608.449,Z 476.894,A -85,B 0,C 180,E1 -446.357,E2 -446.357} C_VEL
LIN {X 0,Y 608.425,Z 479.808,A -85,B 0,C 180,E1 -447.351,E2 -447.351} C_VEL
LIN {X 0,Y 608.442,Z 481.2,A -85,B 0,C 180,E1 -448.014,E2 -448.014} C_VEL
LIN {X 0,Y 608.439,Z 482.783,A -85,B 0,C 180,E1 -449.338,E2 -449.338} C_VEL
LIN {X 0,Y 608.434,Z 483,A -85,B 0,C 180,E1 -449.999,E2 -449.999} C_VEL
LIN {X 0,Y 608.448,Z 482.184,A -85,B 0,C 180,E1 -451.323,E2 -451.323} C_VEL
LIN {X 0,Y 608.442,Z 481.202,A -85,B 0,C 180,E1 -451.985,E2 -451.985} C_VEL
LIN {X 0,Y 608.425,Z 479.811,A -85,B 0,C 180,E1 -452.648,E2 -452.648} C_VEL
LIN {X 0,Y 608.449,Z 476.898,A -85,B 0,C 180,E1 -453.642,E2 -453.642} C_VEL
LIN {X 0,Y 608.432,Z 472.952,A -85,B 0,C 180,E1 -454.637,E2 -454.637} C_VEL
LIN {X 0,Y 608.437,Z 466.88,A -85,B 0,C 180,E1 -455.8,E2 -455.8} C_VEL
LIN {X 0,Y 608.461,Z 460.24,A -85,B 0,C 180,E1 -456.799,E2 -456.799} C_VEL
LIN {X 0,Y 608.456,Z 451.995,A -85,B 0,C 180,E1 -457.8,E2 -457.8} C_VEL
LIN {X 0,Y 608.477,Z 441.606,A -85,B 0,C 180,E1 -458.802,E2 -458.802} C_VEL
LIN {X 0,Y 608.486,Z 430.756,A -85,B 0,C 180,E1 -459.64,E2 -459.64} C_VEL
LIN {X 0,Y 608.489,Z 419.785,A -85,B 0,C 180,E1 -460.312,E2 -460.312} C_VEL
LIN {X 0,Y 608.536,Z 407.796,A -85,B 0,C 180,E1 -460.889,E2 -460.889} C_VEL
LIN {X 0,Y 608.533,Z 395.899,A -85,B 0,C 180,E1 -461.322,E2 -461.322} C_VEL
LIN {X 0,Y 608.542,Z 383.547,A -85,B 0,C 180,E1 -461.638,E2 -461.638} C_VEL
LIN {X 0,Y 608.574,Z 367.788,A -85,B 0,C 180,E1 -461.87,E2 -461.87} C_VEL
LIN {X 0,Y 608.547,Z 271.768,A -85,B 0,C 180,E1 -463.014,E2 -463.014} C_VEL
LIN {X 0,Y 608.459,Z 270.656,A -85,B 0,C 180,E1 -463.101,E2 -463.101} C_VEL
LIN {X 0,Y 608.495,Z 250.715,A -85,B 0,C 180,E1 -465.92,E2 -465.92} C_VEL
LIN {X 0,Y 608.517,Z 231.166,A -85,B 0,C 180,E1 -468.727,E2 -468.727} C_VEL
LIN {X 0,Y 608.549,Z 212.103,A -85,B 0,C 180,E1 -471.51,E2 -471.51} C_VEL
LIN {X 0,Y 608.478,Z 211.266,A -85,B 0,C 180,E1 -471.69,E2 -471.69} C_VEL
LIN {X 0,Y 608.444,Z 211.188,A -85,B 0,C 180,E1 -474.571,E2 -474.571} C_VEL
LIN {X 0,Y 608.486,Z 211.185,A -85,B 0,C 180,E1 -477.208,E2 -477.208} C_VEL
LIN {X 0,Y 608.452,Z 211.196,A -85,B 0,C 180,E1 -479.968,E2 -479.968} C_VEL
LIN {X 0,Y 608.438,Z 211.19,A -85,B 0,C 180,E1 -482.518,E2 -482.518} C_VEL
LIN {X 0,Y 608.426,Z 211.19,A -85,B 0,C 180,E1 -484.901,E2 -484.901} C_VEL
LIN {X 0,Y 608.468,Z 211.19,A -85,B 0,C 180,E1 -487.745,E2 -487.745} C_VEL
LIN {X 0,Y 608.442,Z 211.196,A -85,B 0,C 180,E1 -490.327,E2 -490.327} C_VEL
LIN {X 0,Y 608.419,Z 211.191,A -85,B 0,C 180,E1 -492.962,E2 -492.962} C_VEL
LIN {X 0,Y 608.46,Z 211.188,A -85,B 0,C 180,E1 -495.735,E2 -495.735} C_VEL
LIN {X 0,Y 608.443,Z 211.194,A -85,B 0,C 180,E1 -498.658,E2 -498.658} C_VEL
LIN {X 0,Y 608.41,Z 211.191,A -85,B 0,C 180,E1 -501.406,E2 -501.406} C_VEL
LIN {X 0,Y 608.446,Z 211.189,A -85,B 0,C 180,E1 -503.953,E2 -503.953} C_VEL
LIN {X 0,Y 608.463,Z 211.191,A -85,B 0,C 180,E1 -506.328,E2 -506.328} C_VEL
LIN {X 0,Y 608.442,Z 211.198,A -85,B 0,C 180,E1 -508.731,E2 -508.731} C_VEL
LIN {X 0,Y 608.43,Z 211.191,A -85,B 0,C 180,E1 -511.385,E2 -511.385} C_VEL
LIN {X 0,Y 608.419,Z 211.194,A -85,B 0,C 180,E1 -513.223,E2 -513.223} C_VEL
LIN {X 0,Y 608.422,Z 211.192,A -85,B 0,C 180,E1 -515.426,E2 -515.426} C_VEL
LIN {X 0,Y 608.446,Z 211.189,A -85,B 0,C 180,E1 -518.306,E2 -518.306} C_VEL
LIN {X 0,Y 608.449,Z 211.193,A -85,B 0,C 180,E1 -521.287,E2 -521.287} C_VEL
LIN {X 0,Y 608.406,Z 211.193,A -85,B 0,C 180,E1 -523.903,E2 -523.903} C_VEL
LIN {X 0,Y 608.435,Z 211.191,A -85,B 0,C 180,E1 -526.641,E2 -526.641} C_VEL
LIN {X 0,Y 608.45,Z 211.197,A -85,B 0,C 180,E1 -529.348,E2 -529.348} C_VEL
LIN {X 0,Y 608.392,Z 211.195,A -85,B 0,C 180,E1 -532.03,E2 -532.03} C_VEL
LIN {X 0,Y 608.4,Z 211.194,A -85,B 0,C 180,E1 -534.03,E2 -534.03} C_VEL
LIN {X 0,Y 608.393,Z 211.196,A -85,B 0,C 180,E1 -536.024,E2 -536.024} C_VEL
LIN {X 0,Y 608.401,Z 211.196,A -85,B 0,C 180,E1 -538.012,E2 -538.012} C_VEL
LIN {X 0,Y 608.429,Z 211.193,A -85,B 0,C 180,E1 -539.998,E2 -539.998} C_VEL
LIN {X 0,Y 608.402,Z 211.193,A -85,B 0,C 180,E1 -542.646,E2 -542.646} C_VEL
LIN {X 0,Y 608.415,Z 211.195,A -85,B 0,C 180,E1 -545.3,E2 -545.3} C_VEL
LIN {X 0,Y 608.457,Z 211.194,A -85,B 0,C 180,E1 -547.965,E2 -547.965} C_VEL
LIN {X 0,Y 608.417,Z 211.194,A -85,B 0,C 180,E1 -549.403,E2 -549.403} C_VEL
LIN {X 0,Y 607.767,Z 211.281,A -85,B 0,C 180,E1 -549.955,E2 -549.955} C_VEL
LIN {X 0,Y 604.936,Z 211.635,A -85,B 0,C 180,E1 -550.852,E2 -550.852} C_VEL
LIN {X 0,Y 602.523,Z 211.936,A -85,B 0,C 180,E1 -551.573,E2 -551.573} C_VEL
LIN {X 0,Y 601.465,Z 212.065,A -85,B 0,C 180,E1 -552.13,E2 -552.13} C_VEL
LIN {X 0,Y 601.368,Z 212.073,A -85,B 0,C 180,E1 -552.318,E2 -552.318} C_VEL
LIN {X 0,Y 601.361,Z 212.07,A -85,B 0,C 180,E1 -554.896,E2 -554.896} C_VEL
LIN {X 0,Y 601.355,Z 212.07,A -85,B 0,C 180,E1 -556.985,E2 -556.985} C_VEL
LIN {X 0,Y 601.383,Z 212.067,A -85,B 0,C 180,E1 -559.097,E2 -559.097} C_VEL
LIN {X 0,Y 601.368,Z 212.069,A -85,B 0,C 180,E1 -561.238,E2 -561.238} C_VEL
LIN {X 0,Y 601.441,Z 212.069,A -85,B 0,C 180,E1 -564.138,E2 -564.138} C_VEL
LIN {X 0,Y 601.393,Z 212.066,A -85,B 0,C 180,E1 -567.11,E2 -567.11} C_VEL
LIN {X 0,Y 601.38,Z 212.067,A -85,B 0,C 180,E1 -569.392,E2 -569.392} C_VEL
LIN {X 0,Y 601.373,Z 212.069,A -85,B 0,C 180,E1 -571.725,E2 -571.725} C_VEL
LIN {X 0,Y 601.4,Z 212.069,A -85,B 0,C 180,E1 -574.116,E2 -574.116} C_VEL
LIN {X 0,Y 601.389,Z 212.078,A -85,B 0,C 180,E1 -576.58,E2 -576.58} C_VEL
LIN {X 0,Y 601.41,Z 212.064,A -85,B 0,C 180,E1 -579.534,E2 -579.534} C_VEL
LIN {X 0,Y 601.388,Z 212.067,A -85,B 0,C 180,E1 -581.763,E2 -581.763} C_VEL
LIN {X 0,Y 601.392,Z 212.073,A -85,B 0,C 180,E1 -584.533,E2 -584.533} C_VEL
LIN {X 0,Y 601.462,Z 212.292,A -85,B 0,C 180,E1 -586.793,E2 -586.793} C_VEL
LIN {X 0,Y 601.497,Z 225.601,A -85,B 0,C 180,E1 -588.949,E2 -588.949} C_VEL
LIN {X 0,Y 601.454,Z 243.17,A -85,B 0,C 180,E1 -591.736,E2 -591.736} C_VEL
LIN {X 0,Y 601.427,Z 256.886,A -85,B 0,C 180,E1 -593.854,E2 -593.854} C_VEL
LIN {X 0,Y 601.62,Z 259.959,A -85,B 0,C 180,E1 -593.924,E2 -593.924} C_VEL
LIN {X 0,Y 601.623,Z 364.635,A -85,B 0,C 180,E1 -595.198,E2 -595.198} C_VEL
LIN {X 0,Y 601.58,Z 378.269,A -85,B 0,C 180,E1 -595.513,E2 -595.513} C_VEL
LIN {X 0,Y 601.56,Z 390.883,A -85,B 0,C 180,E1 -595.946,E2 -595.946} C_VEL
LIN {X 0,Y 601.495,Z 402.573,A -85,B 0,C 180,E1 -596.491,E2 -596.491} C_VEL
LIN {X 0,Y 601.461,Z 414.006,A -85,B 0,C 180,E1 -597.174,E2 -597.174} C_VEL
LIN {X 0,Y 601.427,Z 424.783,A -85,B 0,C 180,E1 -597.98,E2 -597.98} C_VEL
LIN {X 0,Y 601.404,Z 434.452,A -85,B 0,C 180,E1 -598.888,E2 -598.888} C_VEL
LIN {X 0,Y 601.397,Z 442.858,A -85,B 0,C 180,E1 -599.849,E2 -599.849} C_VEL
LIN {X 0,Y 601.368,Z 450.453,A -85,B 0,C 180,E1 -600.938,E2 -600.938} C_VEL
LIN {X 0,Y 601.347,Z 456.91,A -85,B 0,C 180,E1 -602.13,E2 -602.13} C_VEL
LIN {X 0,Y 601.351,Z 461.547,A -85,B 0,C 180,E1 -603.26,E2 -603.26} C_VEL
LIN {X 0,Y 601.327,Z 464.842,A -85,B 0,C 180,E1 -604.379,E2 -604.379} C_VEL
LIN {X 0,Y 601.342,Z 466.34,A -85,B 0,C 180,E1 -605.12,E2 -605.12} C_VEL
LIN {X 0,Y 601.345,Z 467.359,A -85,B 0,C 180,E1 -605.856,E2 -605.856} C_VEL
LIN {X 0,Y 601.321,Z 467.9,A -85,B 0,C 180,E1 -606.586,E2 -606.586} C_VEL
LIN {X 0,Y 601.347,Z 467.924,A -85,B 0,C 180,E1 -607.4,E2 -607.4} C_VEL
LIN {X 0,Y 601.333,Z 467.558,A -85,B 0,C 180,E1 -608.039,E2 -608.039} C_VEL
LIN {X 0,Y 601.354,Z 465.923,A -85,B 0,C 180,E1 -609.21,E2 -609.21} C_VEL
LIN {X 0,Y 601.34,Z 462.485,A -85,B 0,C 180,E1 -610.545,E2 -610.545} C_VEL
LIN {X 0,Y 601.345,Z 458.505,A -85,B 0,C 180,E1 -611.607,E2 -611.607} C_VEL
LIN {X 0,Y 601.374,Z 453.315,A -85,B 0,C 180,E1 -612.663,E2 -612.663} C_VEL
LIN {X 0,Y 601.373,Z 446.786,A -85,B 0,C 180,E1 -613.712,E2 -613.712} C_VEL
LIN {X 0,Y 601.394,Z 438.585,A -85,B 0,C 180,E1 -614.756,E2 -614.756} C_VEL
LIN {X 0,Y 601.442,Z 428.386,A -85,B 0,C 180,E1 -615.796,E2 -615.796} C_VEL
LIN {X 0,Y 601.441,Z 417.721,A -85,B 0,C 180,E1 -616.657,E2 -616.657} C_VEL
LIN {X 0,Y 601.48,Z 407.154,A -85,B 0,C 180,E1 -617.345,E2 -617.345} C_VEL
LIN {X 0,Y 601.53,Z 395.483,A -85,B 0,C 180,E1 -617.946,E2 -617.946} C_VEL
LIN {X 0,Y 601.571,Z 383.411,A -85,B 0,C 180,E1 -618.417,E2 -618.417} C_VEL
LIN {X 0,Y 601.618,Z 370.128,A -85,B 0,C 180,E1 -618.784,E2 -618.784} C_VEL
LIN {X 0,Y 601.622,Z 356.787,A -85,B 0,C 180,E1 -619.006,E2 -619.006} C_VEL
LIN {X 0,Y 601.473,Z 257.547,A -85,B 0,C 180,E1 -620.204,E2 -620.204} C_VEL
LIN {X 0,Y 601.408,Z 256.401,A -85,B 0,C 180,E1 -620.288,E2 -620.288} C_VEL
LIN {X 0,Y 601.468,Z 238.307,A -85,B 0,C 180,E1 -623.122,E2 -623.122} C_VEL
LIN {X 0,Y 601.537,Z 220.356,A -85,B 0,C 180,E1 -625.981,E2 -625.981} C_VEL
LIN {X 0,Y 601.451,Z 212.2,A -85,B 0,C 180,E1 -627.322,E2 -627.322} C_VEL
LIN {X 0,Y 601.388,Z 212.068,A -85,B 0,C 180,E1 -630.001,E2 -630.001} C_VEL
LIN {X 0,Y 601.401,Z 212.066,A -85,B 0,C 180,E1 -632.68,E2 -632.68} C_VEL
LIN {X 0,Y 601.422,Z 212.072,A -85,B 0,C 180,E1 -635.365,E2 -635.365} C_VEL
LIN {X 0,Y 601.4,Z 212.068,A -85,B 0,C 180,E1 -638.062,E2 -638.062} C_VEL
LIN {X 0,Y 601.363,Z 212.07,A -85,B 0,C 180,E1 -640.778,E2 -640.778} C_VEL
LIN {X 0,Y 601.387,Z 212.074,A -85,B 0,C 180,E1 -643.517,E2 -643.517} C_VEL
LIN {X 0,Y 601.387,Z 212.07,A -85,B 0,C 180,E1 -646.289,E2 -646.289} C_VEL
LIN {X 0,Y 601.375,Z 212.068,A -85,B 0,C 180,E1 -649.101,E2 -649.101} C_VEL
LIN {X 0,Y 601.384,Z 212.078,A -85,B 0,C 180,E1 -651.961,E2 -651.961} C_VEL
LIN {X 0,Y 601.42,Z 212.069,A -85,B 0,C 180,E1 -654.299,E2 -654.299} C_VEL
LIN {X 0,Y 601.353,Z 212.071,A -85,B 0,C 180,E1 -657.116,E2 -657.116} C_VEL
LIN {X 0,Y 601.359,Z 212.07,A -85,B 0,C 180,E1 -659.397,E2 -659.397} C_VEL
LIN {X 0,Y 601.37,Z 212.071,A -85,B 0,C 180,E1 -661.729,E2 -661.729} C_VEL
LIN {X 0,Y 601.387,Z 212.073,A -85,B 0,C 180,E1 -664.121,E2 -664.121} C_VEL
LIN {X 0,Y 601.36,Z 212.079,A -85,B 0,C 180,E1 -666.586,E2 -666.586} C_VEL
LIN {X 0,Y 601.355,Z 212.073,A -85,B 0,C 180,E1 -669.131,E2 -669.131} C_VEL
LIN {X 0,Y 601.37,Z 212.068,A -85,B 0,C 180,E1 -671.77,E2 -671.77} C_VEL
LIN {X 0,Y 601.372,Z 212.076,A -85,B 0,C 180,E1 -674.535,E2 -674.535} C_VEL
LIN {X 0,Y 601.405,Z 212.069,A -85,B 0,C 180,E1 -676.43,E2 -676.43} C_VEL
LIN {X 0,Y 601.365,Z 212.071,A -85,B 0,C 180,E1 -679.433,E2 -679.433} C_VEL
LIN {X 0,Y 601.361,Z 212.069,A -85,B 0,C 180,E1 -681.732,E2 -681.732} C_VEL
LIN {X 0,Y 601.35,Z 212.071,A -85,B 0,C 180,E1 -684.247,E2 -684.247} C_VEL
LIN {X 0,Y 601.374,Z 212.072,A -85,B 0,C 180,E1 -686.687,E2 -686.687} C_VEL
LIN {X 0,Y 601.382,Z 212.076,A -85,B 0,C 180,E1 -689.06,E2 -689.06} C_VEL
LIN {X 0,Y 601.421,Z 212.071,A -85,B 0,C 180,E1 -691.376,E2 -691.376} C_VEL
LIN {X 0,Y 601.36,Z 212.069,A -85,B 0,C 180,E1 -694.383,E2 -694.383} C_VEL
LIN {X 0,Y 601.354,Z 212.071,A -85,B 0,C 180,E1 -696.59,E2 -696.59} C_VEL
LIN {X 0,Y 601.422,Z 212.073,A -85,B 0,C 180,E1 -699.481,E2 -699.481} C_VEL
LIN {X 0,Y 601.359,Z 212.07,A -85,B 0,C 180,E1 -702.314,E2 -702.314} C_VEL
LIN {X 0,Y 601.376,Z 212.068,A -85,B 0,C 180,E1 -704.411,E2 -704.411} C_VEL
LIN {X 0,Y 601.382,Z 212.068,A -85,B 0,C 180,E1 -706.486,E2 -706.486} C_VEL
LIN {X 0,Y 601.348,Z 212.072,A -85,B 0,C 180,E1 -709.026,E2 -709.026} C_VEL
LIN {X 0,Y 601.378,Z 212.069,A -85,B 0,C 180,E1 -711.264,E2 -711.264} C_VEL
LIN {X 0,Y 601.409,Z 212.074,A -85,B 0,C 180,E1 -713.965,E2 -713.965} C_VEL
LIN {X 0,Y 601.377,Z 212.069,A -85,B 0,C 180,E1 -716.653,E2 -716.653} C_VEL
LIN {X 0,Y 601.406,Z 212.067,A -85,B 0,C 180,E1 -718.663,E2 -718.663} C_VEL
LIN {X 0,Y 601.442,Z 212.063,A -85,B 0,C 180,E1 -720.672,E2 -720.672} C_VEL
LIN {X 0,Y 601.359,Z 212.069,A -85,B 0,C 180,E1 -723.352,E2 -723.352} C_VEL
LIN {X 0,Y 601.389,Z 212.065,A -85,B 0,C 180,E1 -725.367,E2 -725.367} C_VEL
LIN {X 0,Y 601.372,Z 212.068,A -85,B 0,C 180,E1 -727.388,E2 -727.388} C_VEL
LIN {X 0,Y 601.386,Z 212.067,A -85,B 0,C 180,E1 -729.418,E2 -729.418} C_VEL
LIN {X 0,Y 601.403,Z 212.064,A -85,B 0,C 180,E1 -731.461,E2 -731.461} C_VEL
LIN {X 0,Y 601.406,Z 212.068,A -85,B 0,C 180,E1 -734.208,E2 -734.208} C_VEL
LIN {X 0,Y 601.414,Z 212.07,A -85,B 0,C 180,E1 -736.988,E2 -736.988} C_VEL
LIN {X 0,Y 601.387,Z 212.066,A -85,B 0,C 180,E1 -739.812,E2 -739.812} C_VEL
LIN {X 0,Y 601.41,Z 212.069,A -85,B 0,C 180,E1 -742.604,E2 -742.604} C_VEL
LIN {X 0,Y 601.431,Z 212.063,A -85,B 0,C 180,E1 -745.619,E2 -745.619} C_VEL
LIN {X 0,Y 601.374,Z 212.069,A -85,B 0,C 180,E1 -747.871,E2 -747.871} C_VEL
LIN {X 0,Y 601.406,Z 212.064,A -85,B 0,C 180,E1 -750.167,E2 -750.167} C_VEL
LIN {X 0,Y 601.401,Z 212.067,A -85,B 0,C 180,E1 -752.712,E2 -752.712} C_VEL
LIN {X 0,Y 601.382,Z 212.075,A -85,B 0,C 180,E1 -755.11,E2 -755.11} C_VEL
LIN {X 0,Y 601.437,Z 212.071,A -85,B 0,C 180,E1 -757.42,E2 -757.42} C_VEL
LIN {X 0,Y 601.407,Z 212.067,A -85,B 0,C 180,E1 -759.997,E2 -759.997} C_VEL
LIN {X 0,Y 601.38,Z 212.067,A -85,B 0,C 180,E1 -762.674,E2 -762.674} C_VEL
LIN {X 0,Y 601.407,Z 212.072,A -85,B 0,C 180,E1 -765.48,E2 -765.48} C_VEL
LIN {X 0,Y 601.421,Z 212.064,A -85,B 0,C 180,E1 -768.408,E2 -768.408} C_VEL
LIN {X 0,Y 601.397,Z 212.065,A -85,B 0,C 180,E1 -770.872,E2 -770.872} C_VEL
LIN {X 0,Y 601.392,Z 212.069,A -85,B 0,C 180,E1 -773.416,E2 -773.416} C_VEL
LIN {X 0,Y 601.436,Z 212.071,A -85,B 0,C 180,E1 -776.065,E2 -776.065} C_VEL
LIN {X 0,Y 601.406,Z 212.064,A -85,B 0,C 180,E1 -779.057,E2 -779.057} C_VEL
LIN {X 0,Y 601.413,Z 212.064,A -85,B 0,C 180,E1 -781.372,E2 -781.372} C_VEL
LIN {X 0,Y 601.398,Z 212.067,A -85,B 0,C 180,E1 -783.636,E2 -783.636} C_VEL
LIN {X 0,Y 601.418,Z 212.071,A -85,B 0,C 180,E1 -786.589,E2 -786.589} C_VEL
LIN {X 0,Y 601.452,Z 212.24,A -85,B 0,C 180,E1 -788.222,E2 -788.222} C_VEL
LIN {X 0,Y 601.611,Z 218.34,A -85,B 0,C 180,E1 -789.158,E2 -789.158} C_VEL
LIN {X 0,Y 601.529,Z 237.434,A -85,B 0,C 180,E1 -791.964,E2 -791.964} C_VEL
LIN {X 0,Y 601.45,Z 255.533,A -85,B 0,C 180,E1 -794.583,E2 -794.583} C_VEL
LIN {X 0,Y 601.461,Z 271.278,A -85,B 0,C 180,E1 -796.807,E2 -796.807} C_VEL
LIN {X 0,Y 601.67,Z 274.681,A -85,B 0,C 180,E1 -796.876,E2 -796.876} C_VEL
LIN {X 0,Y 601.62,Z 378.921,A -85,B 0,C 180,E1 -798.139,E2 -798.139} C_VEL
LIN {X 0,Y 601.592,Z 392.201,A -85,B 0,C 180,E1 -798.438,E2 -798.438} C_VEL
LIN {X 0,Y 601.55,Z 403.922,A -85,B 0,C 180,E1 -798.826,E2 -798.826} C_VEL
LIN {X 0,Y 601.531,Z 414.914,A -85,B 0,C 180,E1 -799.311,E2 -799.311} C_VEL
LIN {X 0,Y 601.462,Z 425.573,A -85,B 0,C 180,E1 -799.905,E2 -799.905} C_VEL
LIN {X 0,Y 601.447,Z 436.47,A -85,B 0,C 180,E1 -800.669,E2 -800.669} C_VEL
LIN {X 0,Y 601.423,Z 445.314,A -85,B 0,C 180,E1 -801.431,E2 -801.431} C_VEL
LIN {X 0,Y 601.396,Z 453.473,A -85,B 0,C 180,E1 -802.276,E2 -802.276} C_VEL
LIN {X 0,Y 601.383,Z 461.467,A -85,B 0,C 180,E1 -803.288,E2 -803.288} C_VEL
LIN {X 0,Y 601.372,Z 467.863,A -85,B 0,C 180,E1 -804.299,E2 -804.299} C_VEL
LIN {X 0,Y 601.336,Z 472.948,A -85,B 0,C 180,E1 -805.307,E2 -805.307} C_VEL
LIN {X 0,Y 601.367,Z 476.894,A -85,B 0,C 180,E1 -806.314,E2 -806.314} C_VEL
LIN {X 0,Y 601.325,Z 479.808,A -85,B 0,C 180,E1 -807.32,E2 -807.32} C_VEL
LIN {X 0,Y 601.341,Z 481.201,A -85,B 0,C 180,E1 -807.99,E2 -807.99} C_VEL
LIN {X 0,Y 601.339,Z 482.783,A -85,B 0,C 180,E1 -809.33,E2 -809.33} C_VEL
LIN {X 0,Y 601.335,Z 483,A -85,B 0,C 180,E1 -809.999,E2 -809.999} C_VEL
LIN {X 0,Y 601.347,Z 482.185,A -85,B 0,C 180,E1 -811.339,E2 -811.339} C_VEL
LIN {X 0,Y 601.341,Z 481.203,A -85,B 0,C 180,E1 -812.009,E2 -812.009} C_VEL
LIN {X 0,Y 601.325,Z 479.811,A -85,B 0,C 180,E1 -812.679,E2 -812.679} C_VEL
LIN {X 0,Y 601.367,Z 476.898,A -85,B 0,C 180,E1 -813.685,E2 -813.685} C_VEL
LIN {X 0,Y 601.336,Z 472.952,A -85,B 0,C 180,E1 -814.692,E2 -814.692} C_VEL
LIN {X 0,Y 601.372,Z 466.881,A -85,B 0,C 180,E1 -815.869,E2 -815.869} C_VEL
LIN {X 0,Y 601.381,Z 460.24,A -85,B 0,C 180,E1 -816.879,E2 -816.879} C_VEL
LIN {X 0,Y 601.4,Z 451.995,A -85,B 0,C 180,E1 -817.892,E2 -817.892} C_VEL
LIN {X 0,Y 601.435,Z 441.607,A -85,B 0,C 180,E1 -818.906,E2 -818.906} C_VEL
LIN {X 0,Y 601.472,Z 430.757,A -85,B 0,C 180,E1 -819.754,E2 -819.754} C_VEL
LIN {X 0,Y 601.495,Z 419.788,A -85,B 0,C 180,E1 -820.433,E2 -820.433} C_VEL
LIN {X 0,Y 601.552,Z 407.663,A -85,B 0,C 180,E1 -821.023,E2 -821.023} C_VEL
LIN {X 0,Y 601.578,Z 395.897,A -85,B 0,C 180,E1 -821.455,E2 -821.455} C_VEL
LIN {X 0,Y 601.608,Z 383.545,A -85,B 0,C 180,E1 -821.774,E2 -821.774} C_VEL
LIN {X 0,Y 601.643,Z 367.788,A -85,B 0,C 180,E1 -822.009,E2 -822.009} C_VEL
LIN {X 0,Y 601.574,Z 272.254,A -85,B 0,C 180,E1 -823.157,E2 -823.157} C_VEL
LIN {X 0,Y 601.453,Z 271.013,A -85,B 0,C 180,E1 -823.213,E2 -823.213} C_VEL
LIN {X 0,Y 601.485,Z 251.921,A -85,B 0,C 180,E1 -825.936,E2 -825.936} C_VEL
LIN {X 0,Y 601.531,Z 233.424,A -85,B 0,C 180,E1 -828.622,E2 -828.622} C_VEL
LIN {X 0,Y 601.645,Z 214.517,A -85,B 0,C 180,E1 -831.409,E2 -831.409} C_VEL
LIN {X 0,Y 601.436,Z 212.144,A -85,B 0,C 180,E1 -831.822,E2 -831.822} C_VEL
LIN {X 0,Y 601.406,Z 212.067,A -85,B 0,C 180,E1 -834.285,E2 -834.285} C_VEL
LIN {X 0,Y 601.455,Z 212.06,A -85,B 0,C 180,E1 -837.11,E2 -837.11} C_VEL
LIN {X 0,Y 601.404,Z 212.07,A -85,B 0,C 180,E1 -840.164,E2 -840.164} C_VEL
LIN {X 0,Y 601.406,Z 212.065,A -85,B 0,C 180,E1 -842.712,E2 -842.712} C_VEL
LIN {X 0,Y 601.383,Z 212.067,A -85,B 0,C 180,E1 -845.109,E2 -845.109} C_VEL
LIN {X 0,Y 601.433,Z 212.062,A -85,B 0,C 180,E1 -847.418,E2 -847.418} C_VEL
LIN {X 0,Y 601.401,Z 212.074,A -85,B 0,C 180,E1 -849.995,E2 -849.995} C_VEL
LIN {X 0,Y 601.381,Z 212.071,A -85,B 0,C 180,E1 -852.672,E2 -852.672} C_VEL
LIN {X 0,Y 601.398,Z 212.066,A -85,B 0,C 180,E1 -855.478,E2 -855.478} C_VEL
LIN {X 0,Y 601.417,Z 212.074,A -85,B 0,C 180,E1 -858.406,E2 -858.406} C_VEL
LIN {X 0,Y 601.387,Z 212.07,A -85,B 0,C 180,E1 -860.87,E2 -860.87} C_VEL
LIN {X 0,Y 601.38,Z 212.068,A -85,B 0,C 180,E1 -863.414,E2 -863.414} C_VEL
LIN {X 0,Y 601.426,Z 212.064,A -85,B 0,C 180,E1 -866.064,E2 -866.064} C_VEL
LIN {X 0,Y 601.391,Z 212.071,A -85,B 0,C 180,E1 -869.055,E2 -869.055} C_VEL
LIN {X 0,Y 601.391,Z 212.068,A -85,B 0,C 180,E1 -871.37,E2 -871.37} C_VEL
LIN {X 0,Y 601.376,Z 212.068,A -85,B 0,C 180,E1 -873.633,E2 -873.633} C_VEL
LIN {X 0,Y 601.391,Z 212.066,A -85,B 0,C 180,E1 -875.855,E2 -875.855} C_VEL
LIN {X 0,Y 601.392,Z 212.074,A -85,B 0,C 180,E1 -878.758,E2 -878.758} C_VEL
LIN {X 0,Y 601.368,Z 212.071,A -85,B 0,C 180,E1 -881.605,E2 -881.605} C_VEL
LIN {X 0,Y 601.396,Z 212.067,A -85,B 0,C 180,E1 -883.71,E2 -883.71} C_VEL
LIN {X 0,Y 601.38,Z 212.068,A -85,B 0,C 180,E1 -886.481,E2 -886.481} C_VEL
LIN {X 0,Y 601.409,Z 212.075,A -85,B 0,C 180,E1 -889.222,E2 -889.222} C_VEL
LIN {X 0,Y 601.375,Z 212.07,A -85,B 0,C 180,E1 -891.936,E2 -891.936} C_VEL
LIN {X 0,Y 601.359,Z 212.072,A -85,B 0,C 180,E1 -893.96,E2 -893.96} C_VEL
LIN {X 0,Y 601.351,Z 212.073,A -85,B 0,C 180,E1 -895.977,E2 -895.977} C_VEL
LIN {X 0,Y 601.377,Z 212.071,A -85,B 0,C 180,E1 -897.989,E2 -897.989} C_VEL
LIN {X 0,Y 601.4,Z 212.068,A -85,B 0,C 180,E1 -899.998,E2 -899.998} C_VEL
LIN {X 0,Y 601.373,Z 212.068,A -85,B 0,C 180,E1 -902.677,E2 -902.677} C_VEL
LIN {X 0,Y 601.383,Z 212.072,A -85,B 0,C 180,E1 -905.362,E2 -905.362} C_VEL
LIN {X 0,Y 601.415,Z 212.069,A -85,B 0,C 180,E1 -908.059,E2 -908.059} C_VEL
LIN {X 0,Y 601.34,Z 212.072,A -85,B 0,C 180,E1 -910.775,E2 -910.775} C_VEL
LIN {X 0,Y 601.368,Z 212.073,A -85,B 0,C 180,E1 -912.318,E2 -912.318} C_VEL
LIN {X 0,Y 600.672,Z 212.158,A -85,B 0,C 180,E1 -912.878,E2 -912.878} C_VEL
LIN {X 0,Y 597.814,Z 212.52,A -85,B 0,C 180,E1 -913.786,E2 -913.786} C_VEL
LIN {X 0,Y 595.418,Z 212.814,A -85,B 0,C 180,E1 -914.516,E2 -914.516} C_VEL
LIN {X 0,Y 594.394,Z 212.938,A -85,B 0,C 180,E1 -915.08,E2 -915.08} C_VEL
LIN {X 0,Y 594.311,Z 212.949,A -85,B 0,C 180,E1 -915.271,E2 -915.271} C_VEL
LIN {X 0,Y 594.319,Z 212.955,A -85,B 0,C 180,E1 -917.903,E2 -917.903} C_VEL
LIN {X 0,Y 594.376,Z 212.942,A -85,B 0,C 180,E1 -920.773,E2 -920.773} C_VEL
LIN {X 0,Y 594.348,Z 212.946,A -85,B 0,C 180,E1 -923.702,E2 -923.702} C_VEL
LIN {X 0,Y 594.346,Z 212.948,A -85,B 0,C 180,E1 -926.698,E2 -926.698} C_VEL
LIN {X 0,Y 594.358,Z 212.944,A -85,B 0,C 180,E1 -928.996,E2 -928.996} C_VEL
LIN {X 0,Y 594.348,Z 212.944,A -85,B 0,C 180,E1 -931.64,E2 -931.64} C_VEL
LIN {X 0,Y 594.378,Z 212.951,A -85,B 0,C 180,E1 -934.576,E2 -934.576} C_VEL
LIN {X 0,Y 594.361,Z 212.942,A -85,B 0,C 180,E1 -937.606,E2 -937.606} C_VEL
LIN {X 0,Y 594.345,Z 212.953,A -85,B 0,C 180,E1 -940.564,E2 -940.564} C_VEL
LIN {X 0,Y 594.356,Z 212.946,A -85,B 0,C 180,E1 -943.295,E2 -943.295} C_VEL
LIN {X 0,Y 594.402,Z 212.992,A -85,B 0,C 180,E1 -946.597,E2 -946.597} C_VEL
LIN {X 0,Y 594.593,Z 214.183,A -85,B 0,C 180,E1 -946.872,E2 -946.872} C_VEL
LIN {X 0,Y 594.541,Z 231.346,A -85,B 0,C 180,E1 -949.657,E2 -949.657} C_VEL
LIN {X 0,Y 594.381,Z 248.428,A -85,B 0,C 180,E1 -952.386,E2 -952.386} C_VEL
LIN {X 0,Y 594.41,Z 256.99,A -85,B 0,C 180,E1 -953.702,E2 -953.702} C_VEL
LIN {X 0,Y 594.715,Z 261.09,A -85,B 0,C 180,E1 -953.782,E2 -953.782} C_VEL
LIN {X 0,Y 594.695,Z 364.535,A -85,B 0,C 180,E1 -955.056,E2 -955.056} C_VEL
LIN {X 0,Y 594.624,Z 377.718,A -85,B 0,C 180,E1 -955.36,E2 -955.36} C_VEL
LIN {X 0,Y 594.59,Z 390.065,A -85,B 0,C 180,E1 -955.783,E2 -955.783} C_VEL
LIN {X 0,Y 594.521,Z 402.292,A -85,B 0,C 180,E1 -956.351,E2 -956.351} C_VEL
LIN {X 0,Y 594.445,Z 414.23,A -85,B 0,C 180,E1 -957.071,E2 -957.071} C_VEL
LIN {X 0,Y 594.399,Z 424.594,A -85,B 0,C 180,E1 -957.856,E2 -957.856} C_VEL
LIN {X 0,Y 594.371,Z 433.078,A -85,B 0,C 180,E1 -958.651,E2 -958.651} C_VEL
LIN {X 0,Y 594.316,Z 440.271,A -85,B 0,C 180,E1 -959.438,E2 -959.438} C_VEL
LIN {X 0,Y 594.312,Z 447.566,A -85,B 0,C 180,E1 -960.416,E2 -960.416} C_VEL
LIN {X 0,Y 594.253,Z 453.582,A -85,B 0,C 180,E1 -961.41,E2 -961.41} C_VEL
LIN {X 0,Y 594.25,Z 458.943,A -85,B 0,C 180,E1 -962.534,E2 -962.534} C_VEL
LIN {X 0,Y 594.278,Z 463.02,A -85,B 0,C 180,E1 -963.675,E2 -963.675} C_VEL
LIN {X 0,Y 594.225,Z 465.812,A -85,B 0,C 180,E1 -964.801,E2 -964.801} C_VEL
LIN {X 0,Y 594.239,Z 467.068,A -85,B 0,C 180,E1 -965.588,E2 -965.588} C_VEL
LIN {X 0,Y 594.22,Z 467.731,A -85,B 0,C 180,E1 -966.29,E2 -966.29} C_VEL
LIN {X 0,Y 594.252,Z 467.952,A -85,B 0,C 180,E1 -967.28,E2 -967.28} C_VEL
LIN {X 0,Y 594.215,Z 467.08,A -85,B 0,C 180,E1 -968.492,E2 -968.492} C_VEL
LIN {X 0,Y 594.266,Z 465.954,A -85,B 0,C 180,E1 -969.22,E2 -969.22} C_VEL
LIN {X 0,Y 594.258,Z 463.366,A -85,B 0,C 180,E1 -970.303,E2 -970.303} C_VEL
LIN {X 0,Y 594.26,Z 459.683,A -85,B 0,C 180,E1 -971.379,E2 -971.379} C_VEL
LIN {X 0,Y 594.279,Z 454.812,A -85,B 0,C 180,E1 -972.449,E2 -972.449} C_VEL
LIN {X 0,Y 594.3,Z 448.627,A -85,B 0,C 180,E1 -973.513,E2 -973.513} C_VEL
LIN {X 0,Y 594.352,Z 440.916,A -85,B 0,C 180,E1 -974.571,E2 -974.571} C_VEL
LIN {X 0,Y 594.381,Z 432.984,A -85,B 0,C 180,E1 -975.449,E2 -975.449} C_VEL
LIN {X 0,Y 594.415,Z 424.99,A -85,B 0,C 180,E1 -976.2,E2 -976.2} C_VEL
LIN {X 0,Y 594.444,Z 414.22,A -85,B 0,C 180,E1 -977.019,E2 -977.019} C_VEL
LIN {X 0,Y 594.479,Z 402.764,A -85,B 0,C 180,E1 -977.714,E2 -977.714} C_VEL
LIN {X 0,Y 594.585,Z 390.794,A -85,B 0,C 180,E1 -978.279,E2 -978.279} C_VEL
LIN {X 0,Y 594.649,Z 377.596,A -85,B 0,C 180,E1 -978.733,E2 -978.733} C_VEL
LIN {X 0,Y 594.672,Z 364.033,A -85,B 0,C 180,E1 -979.044,E2 -979.044} C_VEL
LIN {X 0,Y 594.552,Z 258.236,A -85,B 0,C 180,E1 -980.346,E2 -980.346} C_VEL
LIN {X 0,Y 594.381,Z 256.527,A -85,B 0,C 180,E1 -980.429,E2 -980.429} C_VEL
LIN {X 0,Y 594.454,Z 238.855,A -85,B 0,C 180,E1 -983.229,E2 -983.229} C_VEL
LIN {X 0,Y 594.556,Z 221.022,A -85,B 0,C 180,E1 -986.103,E2 -986.103} C_VEL
LIN {X 0,Y 594.414,Z 213.117,A -85,B 0,C 180,E1 -987.417,E2 -987.417} C_VEL
LIN {X 0,Y 594.358,Z 212.944,A -85,B 0,C 180,E1 -990.001,E2 -990.001} C_VEL
LIN {X 0,Y 594.369,Z 212.943,A -85,B 0,C 180,E1 -992.711,E2 -992.711} C_VEL
LIN {X 0,Y 594.38,Z 212.95,A -85,B 0,C 180,E1 -995.428,E2 -995.428} C_VEL
LIN {X 0,Y 594.372,Z 212.942,A -85,B 0,C 180,E1 -998.158,E2 -998.158} C_VEL
LIN {X 0,Y 594.341,Z 212.947,A -85,B 0,C 180,E1 -1001.071,E2 -1001.071} C_VEL
LIN {X 0,Y 594.348,Z 212.954,A -85,B 0,C 180,E1 -1003.68,E2 -1003.68} C_VEL
LIN {X 0,Y 594.326,Z 212.946,A -85,B 0,C 180,E1 -1006.712,E2 -1006.712} C_VEL
LIN {X 0,Y 594.329,Z 212.948,A -85,B 0,C 180,E1 -1009.336,E2 -1009.336} C_VEL
LIN {X 0,Y 594.328,Z 212.949,A -85,B 0,C 180,E1 -1011.505,E2 -1011.505} C_VEL
LIN {X 0,Y 594.355,Z 212.947,A -85,B 0,C 180,E1 -1014.448,E2 -1014.448} C_VEL
LIN {X 0,Y 594.319,Z 212.949,A -85,B 0,C 180,E1 -1016.703,E2 -1016.703} C_VEL
LIN {X 0,Y 594.34,Z 212.944,A -85,B 0,C 180,E1 -1019.001,E2 -1019.001} C_VEL
LIN {X 0,Y 594.341,Z 212.946,A -85,B 0,C 180,E1 -1021.644,E2 -1021.644} C_VEL
LIN {X 0,Y 594.336,Z 212.952,A -85,B 0,C 180,E1 -1024.583,E2 -1024.583} C_VEL
LIN {X 0,Y 594.323,Z 212.946,A -85,B 0,C 180,E1 -1027.606,E2 -1027.606} C_VEL
LIN {X 0,Y 594.331,Z 212.957,A -85,B 0,C 180,E1 -1030.57,E2 -1030.57} C_VEL
LIN {X 0,Y 594.32,Z 212.948,A -85,B 0,C 180,E1 -1033.304,E2 -1033.304} C_VEL
LIN {X 0,Y 594.327,Z 212.948,A -85,B 0,C 180,E1 -1036.165,E2 -1036.165} C_VEL
LIN {X 0,Y 594.342,Z 212.949,A -85,B 0,C 180,E1 -1039.182,E2 -1039.182} C_VEL
LIN {X 0,Y 594.343,Z 212.943,A -85,B 0,C 180,E1 -1042.06,E2 -1042.06} C_VEL
LIN {X 0,Y 594.331,Z 212.95,A -85,B 0,C 180,E1 -1044.68,E2 -1044.68} C_VEL
LIN {X 0,Y 594.355,Z 212.954,A -85,B 0,C 180,E1 -1047.092,E2 -1047.092} C_VEL
LIN {X 0,Y 594.331,Z 212.947,A -85,B 0,C 180,E1 -1049.681,E2 -1049.681} C_VEL
LIN {X 0,Y 594.325,Z 212.948,A -85,B 0,C 180,E1 -1051.774,E2 -1051.774} C_VEL
LIN {X 0,Y 594.325,Z 212.947,A -85,B 0,C 180,E1 -1054.057,E2 -1054.057} C_VEL
LIN {X 0,Y 594.341,Z 212.944,A -85,B 0,C 180,E1 -1056.297,E2 -1056.297} C_VEL
LIN {X 0,Y 594.393,Z 212.944,A -85,B 0,C 180,E1 -1059.227,E2 -1059.227} C_VEL
LIN {X 0,Y 594.322,Z 212.947,A -85,B 0,C 180,E1 -1062.097,E2 -1062.097} C_VEL
LIN {X 0,Y 594.334,Z 212.947,A -85,B 0,C 180,E1 -1064.221,E2 -1064.221} C_VEL
LIN {X 0,Y 594.356,Z 212.944,A -85,B 0,C 180,E1 -1066.323,E2 -1066.323} C_VEL
LIN {X 0,Y 594.326,Z 212.946,A -85,B 0,C 180,E1 -1068.959,E2 -1068.959} C_VEL
LIN {X 0,Y 594.375,Z 212.95,A -85,B 0,C 180,E1 -1071.845,E2 -1071.845} C_VEL
LIN {X 0,Y 594.366,Z 212.942,A -85,B 0,C 180,E1 -1074.574,E2 -1074.574} C_VEL
LIN {X 0,Y 594.365,Z 212.941,A -85,B 0,C 180,E1 -1077.291,E2 -1077.291} C_VEL
LIN {X 0,Y 594.403,Z 212.944,A -85,B 0,C 180,E1 -1080.002,E2 -1080.002} C_VEL
LIN {X 0,Y 594.403,Z 212.939,A -85,B 0,C 180,E1 -1082.713,E2 -1082.713} C_VEL
LIN {X 0,Y 594.356,Z 212.94,A -85,B 0,C 180,E1 -1085.43,E2 -1085.43} C_VEL
LIN {X 0,Y 594.344,Z 212.943,A -85,B 0,C 180,E1 -1087.476,E2 -1087.476} C_VEL
LIN {X 0,Y 594.336,Z 212.945,A -85,B 0,C 180,E1 -1089.531,E2 -1089.531} C_VEL
LIN {X 0,Y 594.372,Z 212.94,A -85,B 0,C 180,E1 -1091.598,E2 -1091.598} C_VEL
LIN {X 0,Y 594.385,Z 212.944,A -85,B 0,C 180,E1 -1094.379,E2 -1094.379} C_VEL
LIN {X 0,Y 594.376,Z 212.943,A -85,B 0,C 180,E1 -1097.196,E2 -1097.196} C_VEL
LIN {X 0,Y 594.358,Z 212.943,A -85,B 0,C 180,E1 -1100.056,E2 -1100.056} C_VEL
LIN {X 0,Y 594.355,Z 212.952,A -85,B 0,C 180,E1 -1102.969,E2 -1102.969} C_VEL
LIN {X 0,Y 594.374,Z 212.94,A -85,B 0,C 180,E1 -1106.02,E2 -1106.02} C_VEL
LIN {X 0,Y 594.33,Z 212.946,A -85,B 0,C 180,E1 -1108.231,E2 -1108.231} C_VEL
LIN {X 0,Y 594.369,Z 212.942,A -85,B 0,C 180,E1 -1110.562,E2 -1110.562} C_VEL
LIN {X 0,Y 594.378,Z 212.945,A -85,B 0,C 180,E1 -1112.952,E2 -1112.952} C_VEL
LIN {X 0,Y 594.332,Z 212.955,A -85,B 0,C 180,E1 -1115.412,E2 -1115.412} C_VEL
LIN {X 0,Y 594.383,Z 212.941,A -85,B 0,C 180,E1 -1117.942,E2 -1117.942} C_VEL
LIN {X 0,Y 594.369,Z 212.942,A -85,B 0,C 180,E1 -1120.821,E2 -1120.821} C_VEL
LIN {X 0,Y 594.35,Z 212.949,A -85,B 0,C 180,E1 -1123.302,E2 -1123.302} C_VEL
LIN {X 0,Y 594.351,Z 212.946,A -85,B 0,C 180,E1 -1126.163,E2 -1126.163} C_VEL
LIN {X 0,Y 594.378,Z 212.94,A -85,B 0,C 180,E1 -1128.536,E2 -1128.536} C_VEL
LIN {X 0,Y 594.375,Z 212.943,A -85,B 0,C 180,E1 -1131.298,E2 -1131.298} C_VEL
LIN {X 0,Y 594.352,Z 212.951,A -85,B 0,C 180,E1 -1133.755,E2 -1133.755} C_VEL
LIN {X 0,Y 594.38,Z 212.946,A -85,B 0,C 180,E1 -1136.239,E2 -1136.239} C_VEL
LIN {X 0,Y 594.372,Z 212.943,A -85,B 0,C 180,E1 -1138.65,E2 -1138.65} C_VEL
LIN {X 0,Y 594.381,Z 212.94,A -85,B 0,C 180,E1 -1141.044,E2 -1141.044} C_VEL
LIN {X 0,Y 594.386,Z 212.939,A -85,B 0,C 180,E1 -1143.3,E2 -1143.3} C_VEL
LIN {X 0,Y 594.356,Z 212.945,A -85,B 0,C 180,E1 -1145.575,E2 -1145.575} C_VEL
LIN {X 0,Y 594.395,Z 213.134,A -85,B 0,C 180,E1 -1148.087,E2 -1148.087} C_VEL
LIN {X 0,Y 594.694,Z 216.84,A -85,B 0,C 180,E1 -1148.678,E2 -1148.678} C_VEL
LIN {X 0,Y 594.574,Z 236.228,A -85,B 0,C 180,E1 -1151.567,E2 -1151.567} C_VEL
LIN {X 0,Y 594.486,Z 254.327,A -85,B 0,C 180,E1 -1154.222,E2 -1154.222} C_VEL
LIN {X 0,Y 594.43,Z 271.271,A -85,B 0,C 180,E1 -1156.648,E2 -1156.648} C_VEL
LIN {X 0,Y 594.768,Z 274.681,A -85,B 0,C 180,E1 -1156.721,E2 -1156.721} C_VEL
LIN {X 0,Y 594.673,Z 378.921,A -85,B 0,C 180,E1 -1157.999,E2 -1157.999} C_VEL
LIN {X 0,Y 594.64,Z 392.201,A -85,B 0,C 180,E1 -1158.301,E2 -1158.301} C_VEL
LIN {X 0,Y 594.589,Z 405.368,A -85,B 0,C 180,E1 -1158.749,E2 -1158.749} C_VEL
LIN {X 0,Y 594.538,Z 416.623,A -85,B 0,C 180,E1 -1159.27,E2 -1159.27} C_VEL
LIN {X 0,Y 594.455,Z 428.193,A -85,B 0,C 180,E1 -1159.957,E2 -1159.957} C_VEL
LIN {X 0,Y 594.414,Z 438.591,A -85,B 0,C 180,E1 -1160.729,E2 -1160.729} C_VEL
LIN {X 0,Y 594.349,Z 447.027,A -85,B 0,C 180,E1 -1161.5,E2 -1161.5} C_VEL
LIN {X 0,Y 594.348,Z 454.956,A -85,B 0,C 180,E1 -1162.355,E2 -1162.355} C_VEL
LIN {X 0,Y 594.281,Z 462.827,A -85,B 0,C 180,E1 -1163.41,E2 -1163.41} C_VEL
LIN {X 0,Y 594.289,Z 469.678,A -85,B 0,C 180,E1 -1164.571,E2 -1164.571} C_VEL
LIN {X 0,Y 594.27,Z 474.369,A -85,B 0,C 180,E1 -1165.591,E2 -1165.591} C_VEL
LIN {X 0,Y 594.267,Z 477.955,A -85,B 0,C 180,E1 -1166.609,E2 -1166.609} C_VEL
LIN {X 0,Y 594.226,Z 479.807,A -85,B 0,C 180,E1 -1167.288,E2 -1167.288} C_VEL
LIN {X 0,Y 594.24,Z 481.2,A -85,B 0,C 180,E1 -1167.966,E2 -1167.966} C_VEL
LIN {X 0,Y 594.239,Z 482.784,A -85,B 0,C 180,E1 -1169.322,E2 -1169.322} C_VEL
LIN {X 0,Y 594.236,Z 483,A -85,B 0,C 180,E1 -1169.999,E2 -1169.999} C_VEL
LIN {X 0,Y 594.247,Z 482.186,A -85,B 0,C 180,E1 -1171.355,E2 -1171.355} C_VEL
LIN {X 0,Y 594.24,Z 481.202,A -85,B 0,C 180,E1 -1172.033,E2 -1172.033} C_VEL
LIN {X 0,Y 594.226,Z 479.811,A -85,B 0,C 180,E1 -1172.711,E2 -1172.711} C_VEL
LIN {X 0,Y 594.289,Z 476.898,A -85,B 0,C 180,E1 -1173.729,E2 -1173.729} C_VEL
LIN {X 0,Y 594.241,Z 472.952,A -85,B 0,C 180,E1 -1174.748,E2 -1174.748} C_VEL
LIN {X 0,Y 594.304,Z 466.881,A -85,B 0,C 180,E1 -1175.939,E2 -1175.939} C_VEL
LIN {X 0,Y 594.308,Z 460.241,A -85,B 0,C 180,E1 -1176.961,E2 -1176.961} C_VEL
LIN {X 0,Y 594.359,Z 451.995,A -85,B 0,C 180,E1 -1177.986,E2 -1177.986} C_VEL
LIN {X 0,Y 594.404,Z 441.607,A -85,B 0,C 180,E1 -1179.013,E2 -1179.013} C_VEL
LIN {X 0,Y 594.444,Z 430.757,A -85,B 0,C 180,E1 -1179.87,E2 -1179.87} C_VEL
LIN {X 0,Y 594.508,Z 419.79,A -85,B 0,C 180,E1 -1180.558,E2 -1180.558} C_VEL
LIN {X 0,Y 594.601,Z 407.161,A -85,B 0,C 180,E1 -1181.175,E2 -1181.175} C_VEL
LIN {X 0,Y 594.621,Z 395.895,A -85,B 0,C 180,E1 -1181.591,E2 -1181.591} C_VEL
LIN {X 0,Y 594.661,Z 383.544,A -85,B 0,C 180,E1 -1181.914,E2 -1181.914} C_VEL
LIN {X 0,Y 594.695,Z 367.788,A -85,B 0,C 180,E1 -1182.151,E2 -1182.151} C_VEL
LIN {X 0,Y 594.63,Z 272.987,A -85,B 0,C 180,E1 -1183.302,E2 -1183.302} C_VEL
LIN {X 0,Y 594.424,Z 271.009,A -85,B 0,C 180,E1 -1183.372,E2 -1183.372} C_VEL
LIN {X 0,Y 594.49,Z 251.921,A -85,B 0,C 180,E1 -1186.129,E2 -1186.129} C_VEL
LIN {X 0,Y 594.594,Z 233.254,A -85,B 0,C 180,E1 -1188.873,E2 -1188.873} C_VEL
LIN {X 0,Y 594.698,Z 215.723,A -85,B 0,C 180,E1 -1191.49,E2 -1191.49} C_VEL
LIN {X 0,Y 594.379,Z 213.027,A -85,B 0,C 180,E1 -1191.958,E2 -1191.958} C_VEL
LIN {X 0,Y 594.368,Z 212.943,A -85,B 0,C 180,E1 -1194.446,E2 -1194.446} C_VEL
LIN {X 0,Y 594.385,Z 212.94,A -85,B 0,C 180,E1 -1196.699,E2 -1196.699} C_VEL
LIN {X 0,Y 594.376,Z 212.941,A -85,B 0,C 180,E1 -1198.998,E2 -1198.998} C_VEL
LIN {X 0,Y 594.39,Z 212.945,A -85,B 0,C 180,E1 -1201.643,E2 -1201.643} C_VEL
LIN {X 0,Y 594.369,Z 212.943,A -85,B 0,C 180,E1 -1204.58,E2 -1204.58} C_VEL
LIN {X 0,Y 594.388,Z 212.942,A -85,B 0,C 180,E1 -1207.607,E2 -1207.607} C_VEL
LIN {X 0,Y 594.36,Z 212.946,A -85,B 0,C 180,E1 -1210.567,E2 -1210.567} C_VEL
LIN {X 0,Y 594.345,Z 212.944,A -85,B 0,C 180,E1 -1213.3,E2 -1213.3} C_VEL
LIN {X 0,Y 594.36,Z 212.951,A -85,B 0,C 180,E1 -1216.16,E2 -1216.16} C_VEL
LIN {X 0,Y 594.373,Z 212.949,A -85,B 0,C 180,E1 -1218.534,E2 -1218.534} C_VEL
LIN {X 0,Y 594.363,Z 212.942,A -85,B 0,C 180,E1 -1221.297,E2 -1221.297} C_VEL
LIN {X 0,Y 594.344,Z 212.945,A -85,B 0,C 180,E1 -1223.754,E2 -1223.754} C_VEL
LIN {X 0,Y 594.372,Z 212.945,A -85,B 0,C 180,E1 -1226.237,E2 -1226.237} C_VEL
LIN {X 0,Y 594.362,Z 212.953,A -85,B 0,C 180,E1 -1228.648,E2 -1228.648} C_VEL
LIN {X 0,Y 594.369,Z 212.946,A -85,B 0,C 180,E1 -1231.043,E2 -1231.043} C_VEL
LIN {X 0,Y 594.36,Z 212.945,A -85,B 0,C 180,E1 -1233.298,E2 -1233.298} C_VEL
LIN {X 0,Y 594.331,Z 212.946,A -85,B 0,C 180,E1 -1235.576,E2 -1235.576} C_VEL
LIN {X 0,Y 594.348,Z 212.947,A -85,B 0,C 180,E1 -1238.494,E2 -1238.494} C_VEL
LIN {X 0,Y 594.354,Z 212.947,A -85,B 0,C 180,E1 -1241.38,E2 -1241.38} C_VEL
LIN {X 0,Y 594.366,Z 212.945,A -85,B 0,C 180,E1 -1243.512,E2 -1243.512} C_VEL
LIN {X 0,Y 594.341,Z 212.944,A -85,B 0,C 180,E1 -1246.318,E2 -1246.318} C_VEL
LIN {X 0,Y 594.369,Z 212.949,A -85,B 0,C 180,E1 -1249.093,E2 -1249.093} C_VEL
LIN {X 0,Y 594.333,Z 212.948,A -85,B 0,C 180,E1 -1251.84,E2 -1251.84} C_VEL
LIN {X 0,Y 594.32,Z 212.95,A -85,B 0,C 180,E1 -1253.888,E2 -1253.888} C_VEL
LIN {X 0,Y 594.308,Z 212.951,A -85,B 0,C 180,E1 -1255.929,E2 -1255.929} C_VEL
LIN {X 0,Y 594.352,Z 212.946,A -85,B 0,C 180,E1 -1257.965,E2 -1257.965} C_VEL
LIN {X 0,Y 594.372,Z 212.944,A -85,B 0,C 180,E1 -1259.998,E2 -1259.998} C_VEL
LIN {X 0,Y 594.344,Z 212.944,A -85,B 0,C 180,E1 -1262.709,E2 -1262.709} C_VEL
LIN {X 0,Y 594.35,Z 212.949,A -85,B 0,C 180,E1 -1265.426,E2 -1265.426} C_VEL
LIN {X 0,Y 594.356,Z 212.947,A -85,B 0,C 180,E1 -1268.155,E2 -1268.155} C_VEL
LIN {X 0,Y 594.33,Z 212.946,A -85,B 0,C 180,E1 -1271.049,E2 -1271.049} C_VEL
LIN {X 0,Y 594.349,Z 212.95,A -85,B 0,C 180,E1 -1273.677,E2 -1273.677} C_VEL
LIN {X 0,Y 594.311,Z 212.949,A -85,B 0,C 180,E1 -1275.271,E2 -1275.271} C_VEL
LIN {X 0,Y 593.645,Z 213.04,A -85,B 0,C 180,E1 -1275.836,E2 -1275.836} C_VEL
LIN {X 0,Y 590.789,Z 213.402,A -85,B 0,C 180,E1 -1276.754,E2 -1276.754} C_VEL
LIN {X 0,Y 588.38,Z 213.703,A -85,B 0,C 180,E1 -1277.492,E2 -1277.492} C_VEL
LIN {X 0,Y 587.353,Z 213.826,A -85,B 0,C 180,E1 -1278.062,E2 -1278.062} C_VEL
LIN {X 0,Y 587.274,Z 213.833,A -85,B 0,C 180,E1 -1278.255,E2 -1278.255} C_VEL
LIN {X 0,Y 587.311,Z 213.82,A -85,B 0,C 180,E1 -1281.035,E2 -1281.035} C_VEL
LIN {X 0,Y 587.288,Z 213.823,A -85,B 0,C 180,E1 -1283.257,E2 -1283.257} C_VEL
LIN {X 0,Y 587.294,Z 213.823,A -85,B 0,C 180,E1 -1285.515,E2 -1285.515} C_VEL
LIN {X 0,Y 587.305,Z 213.828,A -85,B 0,C 180,E1 -1288.594,E2 -1288.594} C_VEL
LIN {X 0,Y 587.297,Z 213.825,A -85,B 0,C 180,E1 -1290.965,E2 -1290.965} C_VEL
LIN {X 0,Y 587.303,Z 213.822,A -85,B 0,C 180,E1 -1293.395,E2 -1293.395} C_VEL
LIN {X 0,Y 587.317,Z 213.821,A -85,B 0,C 180,E1 -1295.894,E2 -1295.894} C_VEL
LIN {X 0,Y 587.306,Z 213.829,A -85,B 0,C 180,E1 -1298.477,E2 -1298.477} C_VEL
LIN {X 0,Y 587.31,Z 213.825,A -85,B 0,C 180,E1 -1301.154,E2 -1301.154} C_VEL
LIN {X 0,Y 587.303,Z 213.824,A -85,B 0,C 180,E1 -1304.112,E2 -1304.112} C_VEL
LIN {X 0,Y 587.386,Z 213.993,A -85,B 0,C 180,E1 -1306.564,E2 -1306.564} C_VEL
LIN {X 0,Y 587.622,Z 217.986,A -85,B 0,C 180,E1 -1307.252,E2 -1307.252} C_VEL
LIN {X 0,Y 587.449,Z 235.563,A -85,B 0,C 180,E1 -1310.128,E2 -1310.128} C_VEL
LIN {X 0,Y 587.355,Z 250.934,A -85,B 0,C 180,E1 -1312.61,E2 -1312.61} C_VEL
LIN {X 0,Y 587.39,Z 256.753,A -85,B 0,C 180,E1 -1313.522,E2 -1313.522} C_VEL
LIN {X 0,Y 587.691,Z 259.227,A -85,B 0,C 180,E1 -1313.598,E2 -1313.598} C_VEL
LIN {X 0,Y 587.749,Z 364.156,A -85,B 0,C 180,E1 -1314.905,E2 -1314.905} C_VEL
LIN {X 0,Y 587.681,Z 377.147,A -85,B 0,C 180,E1 -1315.204,E2 -1315.204} C_VEL
LIN {X 0,Y 587.636,Z 388.955,A -85,B 0,C 180,E1 -1315.604,E2 -1315.604} C_VEL
LIN {X 0,Y 587.555,Z 400.034,A -85,B 0,C 180,E1 -1316.104,E2 -1316.104} C_VEL
LIN {X 0,Y 587.46,Z 411.605,A -85,B 0,C 180,E1 -1316.774,E2 -1316.774} C_VEL
LIN {X 0,Y 587.398,Z 421.921,A -85,B 0,C 180,E1 -1317.525,E2 -1317.525} C_VEL
LIN {X 0,Y 587.361,Z 429.962,A -85,B 0,C 180,E1 -1318.233,E2 -1318.233} C_VEL
LIN {X 0,Y 587.292,Z 438.724,A -85,B 0,C 180,E1 -1319.164,E2 -1319.164} C_VEL
LIN {X 0,Y 587.23,Z 446.814,A -85,B 0,C 180,E1 -1320.221,E2 -1320.221} C_VEL
LIN {X 0,Y 587.166,Z 453.867,A -85,B 0,C 180,E1 -1321.396,E2 -1321.396} C_VEL
LIN {X 0,Y 587.176,Z 459.603,A -85,B 0,C 180,E1 -1322.639,E2 -1322.639} C_VEL
LIN {X 0,Y 587.183,Z 463.634,A -85,B 0,C 180,E1 -1323.845,E2 -1323.845} C_VEL
LIN {X 0,Y 587.128,Z 465.187,A -85,B 0,C 180,E1 -1324.475,E2 -1324.475} C_VEL
LIN {X 0,Y 587.156,Z 466.93,A -85,B 0,C 180,E1 -1325.452,E2 -1325.452} C_VEL
LIN {X 0,Y 587.115,Z 467.936,A -85,B 0,C 180,E1 -1326.733,E2 -1326.733} C_VEL
LIN {X 0,Y 587.148,Z 467.907,A -85,B 0,C 180,E1 -1327.479,E2 -1327.479} C_VEL
LIN {X 0,Y 587.133,Z 467.41,A -85,B 0,C 180,E1 -1328.219,E2 -1328.219} C_VEL
LIN {X 0,Y 587.147,Z 466.371,A -85,B 0,C 180,E1 -1328.998,E2 -1328.998} C_VEL
LIN {X 0,Y 587.156,Z 465.029,A -85,B 0,C 180,E1 -1329.69,E2 -1329.69} C_VEL
LIN {X 0,Y 587.164,Z 461.27,A -85,B 0,C 180,E1 -1330.998,E2 -1330.998} C_VEL
LIN {X 0,Y 587.179,Z 456.203,A -85,B 0,C 180,E1 -1332.23,E2 -1332.23} C_VEL
LIN {X 0,Y 587.22,Z 450.401,A -85,B 0,C 180,E1 -1333.308,E2 -1333.308} C_VEL
LIN {X 0,Y 587.268,Z 443.13,A -85,B 0,C 180,E1 -1334.38,E2 -1334.38} C_VEL
LIN {X 0,Y 587.331,Z 435.702,A -85,B 0,C 180,E1 -1335.27,E2 -1335.27} C_VEL
LIN {X 0,Y 587.362,Z 426.737,A -85,B 0,C 180,E1 -1336.155,E2 -1336.155} C_VEL
LIN {X 0,Y 587.451,Z 416.896,A -85,B 0,C 180,E1 -1336.95,E2 -1336.95} C_VEL
LIN {X 0,Y 587.488,Z 406.158,A -85,B 0,C 180,E1 -1337.653,E2 -1337.653} C_VEL
LIN {X 0,Y 587.584,Z 394.122,A -85,B 0,C 180,E1 -1338.269,E2 -1338.269} C_VEL
LIN {X 0,Y 587.657,Z 382.001,A -85,B 0,C 180,E1 -1338.738,E2 -1338.738} C_VEL
LIN {X 0,Y 587.742,Z 369.537,A -85,B 0,C 180,E1 -1339.08,E2 -1339.08} C_VEL
LIN {X 0,Y 587.741,Z 356.423,A -85,B 0,C 180,E1 -1339.298,E2 -1339.298} C_VEL
LIN {X 0,Y 587.687,Z 259.174,A -85,B 0,C 180,E1 -1340.493,E2 -1340.493} C_VEL
LIN {X 0,Y 587.341,Z 256.951,A -85,B 0,C 180,E1 -1340.552,E2 -1340.552} C_VEL
LIN {X 0,Y 587.47,Z 242.821,A -85,B 0,C 180,E1 -1342.784,E2 -1342.784} C_VEL
LIN {X 0,Y 587.519,Z 224.836,A -85,B 0,C 180,E1 -1345.713,E2 -1345.713} C_VEL
LIN {X 0,Y 587.458,Z 214.461,A -85,B 0,C 180,E1 -1347.429,E2 -1347.429} C_VEL
LIN {X 0,Y 587.321,Z 213.876,A -85,B 0,C 180,E1 -1347.6,E2 -1347.6} C_VEL
LIN {X 0,Y 587.328,Z 213.82,A -85,B 0,C 180,E1 -1350.001,E2 -1350.001} C_VEL
LIN {X 0,Y 587.336,Z 213.819,A -85,B 0,C 180,E1 -1352.744,E2 -1352.744} C_VEL
LIN {X 0,Y 587.34,Z 213.828,A -85,B 0,C 180,E1 -1355.494,E2 -1355.494} C_VEL
LIN {X 0,Y 587.325,Z 213.82,A -85,B 0,C 180,E1 -1358.256,E2 -1358.256} C_VEL
LIN {X 0,Y 587.308,Z 213.823,A -85,B 0,C 180,E1 -1361.135,E2 -1361.135} C_VEL
LIN {X 0,Y 587.323,Z 213.828,A -85,B 0,C 180,E1 -1363.847,E2 -1363.847} C_VEL
LIN {X 0,Y 587.297,Z 213.822,A -85,B 0,C 180,E1 -1366.811,E2 -1366.811} C_VEL
LIN {X 0,Y 587.305,Z 213.826,A -85,B 0,C 180,E1 -1369.577,E2 -1369.577} C_VEL
LIN {X 0,Y 587.302,Z 213.824,A -85,B 0,C 180,E1 -1372.516,E2 -1372.516} C_VEL
LIN {X 0,Y 587.311,Z 213.821,A -85,B 0,C 180,E1 -1374.761,E2 -1374.761} C_VEL
LIN {X 0,Y 587.273,Z 213.825,A -85,B 0,C 180,E1 -1377.049,E2 -1377.049} C_VEL
LIN {X 0,Y 587.31,Z 213.819,A -85,B 0,C 180,E1 -1379.382,E2 -1379.382} C_VEL
LIN {X 0,Y 587.312,Z 213.823,A -85,B 0,C 180,E1 -1381.838,E2 -1381.838} C_VEL
LIN {X 0,Y 587.307,Z 213.831,A -85,B 0,C 180,E1 -1384.349,E2 -1384.349} C_VEL
LIN {X 0,Y 587.279,Z 213.824,A -85,B 0,C 180,E1 -1387.613,E2 -1387.613} C_VEL
LIN {X 0,Y 587.274,Z 213.83,A -85,B 0,C 180,E1 -1390.258,E2 -1390.258} C_VEL
LIN {X 0,Y 587.273,Z 213.827,A -85,B 0,C 180,E1 -1393.119,E2 -1393.119} C_VEL
LIN {X 0,Y 587.276,Z 213.825,A -85,B 0,C 180,E1 -1396.05,E2 -1396.05} C_VEL
LIN {X 0,Y 587.307,Z 213.83,A -85,B 0,C 180,E1 -1398.929,E2 -1398.929} C_VEL
LIN {X 0,Y 587.292,Z 213.823,A -85,B 0,C 180,E1 -1401.522,E2 -1401.522} C_VEL
LIN {X 0,Y 587.265,Z 213.825,A -85,B 0,C 180,E1 -1404.102,E2 -1404.102} C_VEL
LIN {X 0,Y 587.313,Z 213.827,A -85,B 0,C 180,E1 -1406.893,E2 -1406.893} C_VEL
LIN {X 0,Y 587.291,Z 213.827,A -85,B 0,C 180,E1 -1409.498,E2 -1409.498} C_VEL
LIN {X 0,Y 587.288,Z 213.83,A -85,B 0,C 180,E1 -1411.405,E2 -1411.405} C_VEL
LIN {X 0,Y 587.28,Z 213.826,A -85,B 0,C 180,E1 -1413.835,E2 -1413.835} C_VEL
LIN {X 0,Y 587.29,Z 213.824,A -85,B 0,C 180,E1 -1416.743,E2 -1416.743} C_VEL
LIN {X 0,Y 587.311,Z 213.827,A -85,B 0,C 180,E1 -1419.698,E2 -1419.698} C_VEL
LIN {X 0,Y 587.28,Z 213.827,A -85,B 0,C 180,E1 -1421.875,E2 -1421.875} C_VEL
LIN {X 0,Y 587.294,Z 213.821,A -85,B 0,C 180,E1 -1424.739,E2 -1424.739} C_VEL
LIN {X 0,Y 587.283,Z 213.823,A -85,B 0,C 180,E1 -1426.86,E2 -1426.86} C_VEL
LIN {X 0,Y 587.317,Z 213.827,A -85,B 0,C 180,E1 -1429.662,E2 -1429.662} C_VEL
LIN {X 0,Y 587.31,Z 213.821,A -85,B 0,C 180,E1 -1432.439,E2 -1432.439} C_VEL
LIN {X 0,Y 587.323,Z 213.816,A -85,B 0,C 180,E1 -1435.198,E2 -1435.198} C_VEL
LIN {X 0,Y 587.361,Z 213.821,A -85,B 0,C 180,E1 -1437.945,E2 -1437.945} C_VEL
LIN {X 0,Y 587.384,Z 213.814,A -85,B 0,C 180,E1 -1440.688,E2 -1440.688} C_VEL
LIN {X 0,Y 587.267,Z 213.824,A -85,B 0,C 180,E1 -1443.433,E2 -1443.433} C_VEL
LIN {X 0,Y 587.324,Z 213.816,A -85,B 0,C 180,E1 -1445.495,E2 -1445.495} C_VEL
LIN {X 0,Y 587.306,Z 213.82,A -85,B 0,C 180,E1 -1447.566,E2 -1447.566} C_VEL
LIN {X 0,Y 587.305,Z 213.829,A -85,B 0,C 180,E1 -1450.343,E2 -1450.343} C_VEL
LIN {X 0,Y 587.304,Z 213.822,A -85,B 0,C 180,E1 -1453.144,E2 -1453.144} C_VEL
LIN {X 0,Y 587.322,Z 213.819,A -85,B 0,C 180,E1 -1455.265,E2 -1455.265} C_VEL
LIN {X 0,Y 587.309,Z 213.821,A -85,B 0,C 180,E1 -1457.409,E2 -1457.409} C_VEL
LIN {X 0,Y 587.306,Z 213.821,A -85,B 0,C 180,E1 -1459.578,E2 -1459.578} C_VEL
LIN {X 0,Y 587.313,Z 213.819,A -85,B 0,C 180,E1 -1461.776,E2 -1461.776} C_VEL
LIN {X 0,Y 587.309,Z 213.826,A -85,B 0,C 180,E1 -1464.762,E2 -1464.762} C_VEL
LIN {X 0,Y 587.333,Z 213.829,A -85,B 0,C 180,E1 -1467.048,E2 -1467.048} C_VEL
LIN {X 0,Y 587.319,Z 213.825,A -85,B 0,C 180,E1 -1469.383,E2 -1469.383} C_VEL
LIN {X 0,Y 587.322,Z 213.82,A -85,B 0,C 180,E1 -1471.832,E2 -1471.832} C_VEL
LIN {X 0,Y 587.336,Z 213.817,A -85,B 0,C 180,E1 -1474.346,E2 -1474.346} C_VEL
LIN {X 0,Y 587.347,Z 213.823,A -85,B 0,C 180,E1 -1477.609,E2 -1477.609} C_VEL
LIN {X 0,Y 587.312,Z 213.821,A -85,B 0,C 180,E1 -1480.256,E2 -1480.256} C_VEL
LIN {X 0,Y 587.296,Z 213.825,A -85,B 0,C 180,E1 -1483.116,E2 -1483.116} C_VEL
LIN {X 0,Y 587.307,Z 213.825,A -85,B 0,C 180,E1 -1486.048,E2 -1486.048} C_VEL
LIN {X 0,Y 587.319,Z 213.819,A -85,B 0,C 180,E1 -1488.841,E2 -1488.841} C_VEL
LIN {X 0,Y 587.325,Z 213.824,A -85,B 0,C 180,E1 -1491.52,E2 -1491.52} C_VEL
LIN {X 0,Y 587.287,Z 213.831,A -85,B 0,C 180,E1 -1494.099,E2 -1494.099} C_VEL
LIN {X 0,Y 587.337,Z 213.819,A -85,B 0,C 180,E1 -1496.603,E2 -1496.603} C_VEL
LIN {X 0,Y 587.328,Z 213.818,A -85,B 0,C 180,E1 -1499.033,E2 -1499.033} C_VEL
LIN {X 0,Y 587.317,Z 213.82,A -85,B 0,C 180,E1 -1501.402,E2 -1501.402} C_VEL
LIN {X 0,Y 587.335,Z 213.821,A -85,B 0,C 180,E1 -1503.825,E2 -1503.825} C_VEL
LIN {X 0,Y 587.311,Z 213.827,A -85,B 0,C 180,E1 -1505.992,E2 -1505.992} C_VEL
LIN {X 0,Y 587.359,Z 214.028,A -85,B 0,C 180,E1 -1507.95,E2 -1507.95} C_VEL
LIN {X 0,Y 587.751,Z 218.354,A -85,B 0,C 180,E1 -1508.645,E2 -1508.645} C_VEL
LIN {X 0,Y 587.587,Z 238.641,A -85,B 0,C 180,E1 -1511.701,E2 -1511.701} C_VEL
LIN {X 0,Y 587.453,Z 256.74,A -85,B 0,C 180,E1 -1514.384,E2 -1514.384} C_VEL
LIN {X 0,Y 587.406,Z 271.264,A -85,B 0,C 180,E1 -1516.486,E2 -1516.486} C_VEL
LIN {X 0,Y 587.868,Z 274.681,A -85,B 0,C 180,E1 -1516.562,E2 -1516.562} C_VEL
LIN {X 0,Y 587.754,Z 378.921,A -85,B 0,C 180,E1 -1517.855,E2 -1517.855} C_VEL
LIN {X 0,Y 587.686,Z 392.202,A -85,B 0,C 180,E1 -1518.16,E2 -1518.16} C_VEL
LIN {X 0,Y 587.604,Z 404.769,A -85,B 0,C 180,E1 -1518.59,E2 -1518.59} C_VEL
LIN {X 0,Y 587.561,Z 416.621,A -85,B 0,C 180,E1 -1519.141,E2 -1519.141} C_VEL
LIN {X 0,Y 587.437,Z 428.195,A -85,B 0,C 180,E1 -1519.836,E2 -1519.836} C_VEL
LIN {X 0,Y 587.392,Z 438.592,A -85,B 0,C 180,E1 -1520.617,E2 -1520.617} C_VEL
LIN {X 0,Y 587.299,Z 447.042,A -85,B 0,C 180,E1 -1521.397,E2 -1521.397} C_VEL
LIN {X 0,Y 587.274,Z 454.956,A -85,B 0,C 180,E1 -1522.262,E2 -1522.262} C_VEL
LIN {X 0,Y 587.231,Z 461.465,A -85,B 0,C 180,E1 -1523.126,E2 -1523.126} C_VEL
LIN {X 0,Y 587.236,Z 467.864,A -85,B 0,C 180,E1 -1524.161,E2 -1524.161} C_VEL
LIN {X 0,Y 587.147,Z 472.948,A -85,B 0,C 180,E1 -1525.193,E2 -1525.193} C_VEL
LIN {X 0,Y 587.213,Z 476.894,A -85,B 0,C 180,E1 -1526.225,E2 -1526.225} C_VEL
LIN {X 0,Y 587.132,Z 479.807,A -85,B 0,C 180,E1 -1527.255,E2 -1527.255} C_VEL
LIN {X 0,Y 587.139,Z 481.199,A -85,B 0,C 180,E1 -1527.942,E2 -1527.942} C_VEL
LIN {X 0,Y 587.14,Z 482.784,A -85,B 0,C 180,E1 -1529.314,E2 -1529.314} C_VEL
LIN {X 0,Y 587.137,Z 483,A -85,B 0,C 180,E1 -1529.999,E2 -1529.999} C_VEL
LIN {X 0,Y 587.147,Z 482.186,A -85,B 0,C 180,E1 -1531.371,E2 -1531.371} C_VEL
LIN {X 0,Y 587.139,Z 481.202,A -85,B 0,C 180,E1 -1532.057,E2 -1532.057} C_VEL
LIN {X 0,Y 587.132,Z 479.811,A -85,B 0,C 180,E1 -1532.744,E2 -1532.744} C_VEL
LIN {X 0,Y 587.212,Z 476.898,A -85,B 0,C 180,E1 -1533.774,E2 -1533.774} C_VEL
LIN {X 0,Y 587.147,Z 472.952,A -85,B 0,C 180,E1 -1534.806,E2 -1534.806} C_VEL
LIN {X 0,Y 587.217,Z 466.881,A -85,B 0,C 180,E1 -1536.011,E2 -1536.011} C_VEL
LIN {X 0,Y 587.245,Z 460.241,A -85,B 0,C 180,E1 -1537.046,E2 -1537.046} C_VEL
LIN {X 0,Y 587.297,Z 451.996,A -85,B 0,C 180,E1 -1538.082,E2 -1538.082} C_VEL
LIN {X 0,Y 587.357,Z 441.608,A -85,B 0,C 180,E1 -1539.122,E2 -1539.122} C_VEL
LIN {X 0,Y 587.44,Z 430.756,A -85,B 0,C 180,E1 -1539.989,E2 -1539.989} C_VEL
LIN {X 0,Y 587.524,Z 419.792,A -85,B 0,C 180,E1 -1540.684,E2 -1540.684} C_VEL
LIN {X 0,Y 587.618,Z 408.202,A -85,B 0,C 180,E1 -1541.264,E2 -1541.264} C_VEL
LIN {X 0,Y 587.686,Z 395.893,A -85,B 0,C 180,E1 -1541.729,E2 -1541.729} C_VEL
LIN {X 0,Y 587.714,Z 383.542,A -85,B 0,C 180,E1 -1542.057,E2 -1542.057} C_VEL
LIN {X 0,Y 587.768,Z 367.788,A -85,B 0,C 180,E1 -1542.297,E2 -1542.297} C_VEL
LIN {X 0,Y 587.683,Z 273.209,A -85,B 0,C 180,E1 -1543.46,E2 -1543.46} C_VEL
LIN {X 0,Y 587.406,Z 271.282,A -85,B 0,C 180,E1 -1543.513,E2 -1543.513} C_VEL
LIN {X 0,Y 587.483,Z 253.128,A -85,B 0,C 180,E1 -1546.148,E2 -1546.148} C_VEL
LIN {X 0,Y 587.607,Z 235.029,A -85,B 0,C 180,E1 -1548.839,E2 -1548.839} C_VEL
LIN {X 0,Y 587.756,Z 216.925,A -85,B 0,C 180,E1 -1551.573,E2 -1551.573} C_VEL
LIN {X 0,Y 587.343,Z 213.908,A -85,B 0,C 180,E1 -1552.096,E2 -1552.096} C_VEL
LIN {X 0,Y 587.317,Z 213.821,A -85,B 0,C 180,E1 -1554.759,E2 -1554.759} C_VEL
LIN {X 0,Y 587.331,Z 213.819,A -85,B 0,C 180,E1 -1557.045,E2 -1557.045} C_VEL
LIN {X 0,Y 587.318,Z 213.823,A -85,B 0,C 180,E1 -1559.38,E2 -1559.38} C_VEL
LIN {X 0,Y 587.351,Z 213.826,A -85,B 0,C 180,E1 -1561.835,E2 -1561.835} C_VEL
LIN {X 0,Y 587.341,Z 213.821,A -85,B 0,C 180,E1 -1564.345,E2 -1564.345} C_VEL
LIN {X 0,Y 587.343,Z 213.819,A -85,B 0,C 180,E1 -1567.607,E2 -1567.607} C_VEL
LIN {X 0,Y 587.308,Z 213.83,A -85,B 0,C 180,E1 -1570.254,E2 -1570.254} C_VEL
LIN {X 0,Y 587.29,Z 213.823,A -85,B 0,C 180,E1 -1573.007,E2 -1573.007} C_VEL
LIN {X 0,Y 587.312,Z 213.826,A -85,B 0,C 180,E1 -1576.047,E2 -1576.047} C_VEL
LIN {X 0,Y 587.329,Z 213.821,A -85,B 0,C 180,E1 -1578.924,E2 -1578.924} C_VEL
LIN {X 0,Y 587.314,Z 213.819,A -85,B 0,C 180,E1 -1581.518,E2 -1581.518} C_VEL
LIN {X 0,Y 587.285,Z 213.827,A -85,B 0,C 180,E1 -1584.098,E2 -1584.098} C_VEL
LIN {X 0,Y 587.333,Z 213.824,A -85,B 0,C 180,E1 -1586.887,E2 -1586.887} C_VEL
LIN {X 0,Y 587.31,Z 213.82,A -85,B 0,C 180,E1 -1589.827,E2 -1589.827} C_VEL
LIN {X 0,Y 587.296,Z 213.825,A -85,B 0,C 180,E1 -1592.315,E2 -1592.315} C_VEL
LIN {X 0,Y 587.299,Z 213.826,A -85,B 0,C 180,E1 -1595.237,E2 -1595.237} C_VEL
LIN {X 0,Y 587.303,Z 213.822,A -85,B 0,C 180,E1 -1598.223,E2 -1598.223} C_VEL
LIN {X 0,Y 587.333,Z 213.826,A -85,B 0,C 180,E1 -1601.149,E2 -1601.149} C_VEL
LIN {X 0,Y 587.289,Z 213.823,A -85,B 0,C 180,E1 -1604.022,E2 -1604.022} C_VEL
LIN {X 0,Y 587.288,Z 213.828,A -85,B 0,C 180,E1 -1606.856,E2 -1606.856} C_VEL
LIN {X 0,Y 587.287,Z 213.827,A -85,B 0,C 180,E1 -1609.657,E2 -1609.657} C_VEL
LIN {X 0,Y 587.293,Z 213.822,A -85,B 0,C 180,E1 -1612.434,E2 -1612.434} C_VEL
LIN {X 0,Y 587.354,Z 213.822,A -85,B 0,C 180,E1 -1615.193,E2 -1615.193} C_VEL
LIN {X 0,Y 587.326,Z 213.822,A -85,B 0,C 180,E1 -1617.94,E2 -1617.94} C_VEL
LIN {X 0,Y 587.343,Z 213.819,A -85,B 0,C 180,E1 -1619.998,E2 -1619.998} C_VEL
LIN {X 0,Y 587.314,Z 213.82,A -85,B 0,C 180,E1 -1622.741,E2 -1622.741} C_VEL
LIN {X 0,Y 587.317,Z 213.826,A -85,B 0,C 180,E1 -1625.491,E2 -1625.491} C_VEL
LIN {X 0,Y 587.311,Z 213.823,A -85,B 0,C 180,E1 -1628.253,E2 -1628.253} C_VEL
LIN {X 0,Y 587.3,Z 213.822,A -85,B 0,C 180,E1 -1631.114,E2 -1631.114} C_VEL
LIN {X 0,Y 587.332,Z 213.827,A -85,B 0,C 180,E1 -1633.843,E2 -1633.843} C_VEL
LIN {X 0,Y 587.275,Z 213.825,A -85,B 0,C 180,E1 -1636.793,E2 -1636.793} C_VEL
LIN {X 0,Y 587.274,Z 213.833,A -85,B 0,C 180,E1 -1638.255,E2 -1638.255} C_VEL
LIN {X 0,Y 586.631,Z 213.908,A -85,B 0,C 180,E1 -1638.827,E2 -1638.827} C_VEL
LIN {X 0,Y 583.825,Z 214.259,A -85,B 0,C 180,E1 -1639.756,E2 -1639.756} C_VEL
LIN {X 0,Y 581.426,Z 214.558,A -85,B 0,C 180,E1 -1640.503,E2 -1640.503} C_VEL
LIN {X 0,Y 580.368,Z 214.686,A -85,B 0,C 180,E1 -1641.079,E2 -1641.079} C_VEL
LIN {X 0,Y 580.267,Z 214.698,A -85,B 0,C 180,E1 -1641.275,E2 -1641.275} C_VEL
LIN {X 0,Y 580.274,Z 214.707,A -85,B 0,C 180,E1 -1644.314,E2 -1644.314} C_VEL
LIN {X 0,Y 580.239,Z 214.707,A -85,B 0,C 180,E1 -1646.622,E2 -1646.622} C_VEL
LIN {X 0,Y 580.273,Z 214.697,A -85,B 0,C 180,E1 -1649.306,E2 -1649.306} C_VEL
LIN {X 0,Y 580.275,Z 214.703,A -85,B 0,C 180,E1 -1652.198,E2 -1652.198} C_VEL
LIN {X 0,Y 580.276,Z 214.705,A -85,B 0,C 180,E1 -1654.693,E2 -1654.693} C_VEL
LIN {X 0,Y 580.271,Z 214.699,A -85,B 0,C 180,E1 -1657.266,E2 -1657.266} C_VEL
LIN {X 0,Y 580.269,Z 214.702,A -85,B 0,C 180,E1 -1660.269,E2 -1660.269} C_VEL
LIN {X 0,Y 580.26,Z 214.709,A -85,B 0,C 180,E1 -1662.703,E2 -1662.703} C_VEL
LIN {X 0,Y 580.243,Z 214.707,A -85,B 0,C 180,E1 -1665.606,E2 -1665.606} C_VEL
LIN {X 0,Y 580.346,Z 214.934,A -85,B 0,C 180,E1 -1666.467,E2 -1666.467} C_VEL
LIN {X 0,Y 580.667,Z 217.768,A -85,B 0,C 180,E1 -1666.968,E2 -1666.968} C_VEL
LIN {X 0,Y 580.499,Z 235.395,A -85,B 0,C 180,E1 -1669.892,E2 -1669.892} C_VEL
LIN {X 0,Y 580.303,Z 252.791,A -85,B 0,C 180,E1 -1672.733,E2 -1672.733} C_VEL
LIN {X 0,Y 580.372,Z 256.988,A -85,B 0,C 180,E1 -1673.374,E2 -1673.374} C_VEL
LIN {X 0,Y 580.935,Z 262.116,A -85,B 0,C 180,E1 -1673.474,E2 -1673.474} C_VEL
LIN {X 0,Y 580.831,Z 364.284,A -85,B 0,C 180,E1 -1674.76,E2 -1674.76} C_VEL
LIN {X 0,Y 580.729,Z 377.526,A -85,B 0,C 180,E1 -1675.071,E2 -1675.071} C_VEL
LIN {X 0,Y 580.666,Z 389.778,A -85,B 0,C 180,E1 -1675.497,E2 -1675.497} C_VEL
LIN {X 0,Y 580.538,Z 401.69,A -85,B 0,C 180,E1 -1676.057,E2 -1676.057} C_VEL
LIN {X 0,Y 580.431,Z 412.858,A -85,B 0,C 180,E1 -1676.734,E2 -1676.734} C_VEL
LIN {X 0,Y 580.357,Z 424.212,A -85,B 0,C 180,E1 -1677.599,E2 -1677.599} C_VEL
LIN {X 0,Y 580.275,Z 432.786,A -85,B 0,C 180,E1 -1678.412,E2 -1678.412} C_VEL
LIN {X 0,Y 580.212,Z 440.725,A -85,B 0,C 180,E1 -1679.31,E2 -1679.31} C_VEL
LIN {X 0,Y 580.163,Z 447.359,A -85,B 0,C 180,E1 -1680.221,E2 -1680.221} C_VEL
LIN {X 0,Y 580.078,Z 454.297,A -85,B 0,C 180,E1 -1681.409,E2 -1681.409} C_VEL
LIN {X 0,Y 580.087,Z 459.619,A -85,B 0,C 180,E1 -1682.589,E2 -1682.589} C_VEL
LIN {X 0,Y 580.109,Z 463.327,A -85,B 0,C 180,E1 -1683.693,E2 -1683.693} C_VEL
LIN {X 0,Y 580.026,Z 466.113,A -85,B 0,C 180,E1 -1684.908,E2 -1684.908} C_VEL
LIN {X 0,Y 580.037,Z 467.205,A -85,B 0,C 180,E1 -1685.673,E2 -1685.673} C_VEL
LIN {X 0,Y 580.05,Z 468,A -85,B 0,C 180,E1 -1687.037,E2 -1687.037} C_VEL
LIN {X 0,Y 580.028,Z 467.65,A -85,B 0,C 180,E1 -1687.938,E2 -1687.938} C_VEL
LIN {X 0,Y 580.04,Z 466.58,A -85,B 0,C 180,E1 -1688.89,E2 -1688.89} C_VEL
LIN {X 0,Y 580.07,Z 463.926,A -85,B 0,C 180,E1 -1690.17,E2 -1690.17} C_VEL
LIN {X 0,Y 580.082,Z 460.464,A -85,B 0,C 180,E1 -1691.274,E2 -1691.274} C_VEL
LIN {X 0,Y 580.1,Z 455.847,A -85,B 0,C 180,E1 -1692.37,E2 -1692.37} C_VEL
LIN {X 0,Y 580.143,Z 449.879,A -85,B 0,C 180,E1 -1693.474,E2 -1693.474} C_VEL
LIN {X 0,Y 580.202,Z 442.547,A -85,B 0,C 180,E1 -1694.545,E2 -1694.545} C_VEL
LIN {X 0,Y 580.283,Z 434.089,A -85,B 0,C 180,E1 -1695.543,E2 -1695.543} C_VEL
LIN {X 0,Y 580.342,Z 424.913,A -85,B 0,C 180,E1 -1696.431,E2 -1696.431} C_VEL
LIN {X 0,Y 580.404,Z 414.65,A -85,B 0,C 180,E1 -1697.234,E2 -1697.234} C_VEL
LIN {X 0,Y 580.514,Z 403.254,A -85,B 0,C 180,E1 -1697.946,E2 -1697.946} C_VEL
LIN {X 0,Y 580.64,Z 392.367,A -85,B 0,C 180,E1 -1698.483,E2 -1698.483} C_VEL
LIN {X 0,Y 580.726,Z 380.683,A -85,B 0,C 180,E1 -1698.924,E2 -1698.924} C_VEL
LIN {X 0,Y 580.785,Z 368.119,A -85,B 0,C 180,E1 -1699.256,E2 -1699.256} C_VEL
LIN {X 0,Y 580.843,Z 352.05,A -85,B 0,C 180,E1 -1699.5,E2 -1699.5} C_VEL
LIN {X 0,Y 580.732,Z 259.531,A -85,B 0,C 180,E1 -1700.653,E2 -1700.653} C_VEL
LIN {X 0,Y 580.343,Z 256.892,A -85,B 0,C 180,E1 -1700.723,E2 -1700.723} C_VEL
LIN {X 0,Y 580.447,Z 239.236,A -85,B 0,C 180,E1 -1703.568,E2 -1703.568} C_VEL
LIN {X 0,Y 580.612,Z 222.354,A -85,B 0,C 180,E1 -1706.357,E2 -1706.357} C_VEL
LIN {X 0,Y 580.615,Z 217.163,A -85,B 0,C 180,E1 -1707.225,E2 -1707.225} C_VEL
LIN {X 0,Y 580.305,Z 214.817,A -85,B 0,C 180,E1 -1707.658,E2 -1707.658} C_VEL
LIN {X 0,Y 580.299,Z 214.696,A -85,B 0,C 180,E1 -1710.001,E2 -1710.001} C_VEL
LIN {X 0,Y 580.304,Z 214.696,A -85,B 0,C 180,E1 -1712.777,E2 -1712.777} C_VEL
LIN {X 0,Y 580.302,Z 214.703,A -85,B 0,C 180,E1 -1715.56,E2 -1715.56} C_VEL
LIN {X 0,Y 580.288,Z 214.696,A -85,B 0,C 180,E1 -1718.357,E2 -1718.357} C_VEL
LIN {X 0,Y 580.26,Z 214.702,A -85,B 0,C 180,E1 -1721.192,E2 -1721.192} C_VEL
LIN {X 0,Y 580.278,Z 214.702,A -85,B 0,C 180,E1 -1724.019,E2 -1724.019} C_VEL
LIN {X 0,Y 580.274,Z 214.696,A -85,B 0,C 180,E1 -1726.915,E2 -1726.915} C_VEL
LIN {X 0,Y 580.265,Z 214.707,A -85,B 0,C 180,E1 -1729.824,E2 -1729.824} C_VEL
LIN {X 0,Y 580.253,Z 214.7,A -85,B 0,C 180,E1 -1732.805,E2 -1732.805} C_VEL
LIN {X 0,Y 580.266,Z 214.697,A -85,B 0,C 180,E1 -1735.082,E2 -1735.082} C_VEL
LIN {X 0,Y 580.246,Z 214.711,A -85,B 0,C 180,E1 -1738.189,E2 -1738.189} C_VEL
LIN {X 0,Y 580.254,Z 214.703,A -85,B 0,C 180,E1 -1740.697,E2 -1740.697} C_VEL
LIN {X 0,Y 580.251,Z 214.699,A -85,B 0,C 180,E1 -1743.316,E2 -1743.316} C_VEL
LIN {X 0,Y 580.198,Z 214.706,A -85,B 0,C 180,E1 -1745.756,E2 -1745.756} C_VEL
LIN {X 0,Y 580.246,Z 214.705,A -85,B 0,C 180,E1 -1748.15,E2 -1748.15} C_VEL
LIN {X 0,Y 580.248,Z 214.705,A -85,B 0,C 180,E1 -1750.848,E2 -1750.848} C_VEL
LIN {X 0,Y 580.211,Z 214.703,A -85,B 0,C 180,E1 -1753.665,E2 -1753.665} C_VEL
LIN {X 0,Y 580.217,Z 214.712,A -85,B 0,C 180,E1 -1756.616,E2 -1756.616} C_VEL
LIN {X 0,Y 580.267,Z 214.702,A -85,B 0,C 180,E1 -1759.159,E2 -1759.159} C_VEL
LIN {X 0,Y 580.26,Z 214.696,A -85,B 0,C 180,E1 -1761.931,E2 -1761.931} C_VEL
LIN {X 0,Y 580.227,Z 214.704,A -85,B 0,C 180,E1 -1764.455,E2 -1764.455} C_VEL
LIN {X 0,Y 580.265,Z 214.706,A -85,B 0,C 180,E1 -1766.978,E2 -1766.978} C_VEL
LIN {X 0,Y 580.252,Z 214.704,A -85,B 0,C 180,E1 -1769.426,E2 -1769.426} C_VEL
LIN {X 0,Y 580.233,Z 214.699,A -85,B 0,C 180,E1 -1772.154,E2 -1772.154} C_VEL
LIN {X 0,Y 580.228,Z 214.705,A -85,B 0,C 180,E1 -1774.92,E2 -1774.92} C_VEL
LIN {X 0,Y 580.273,Z 214.703,A -85,B 0,C 180,E1 -1777.2,E2 -1777.2} C_VEL
LIN {X 0,Y 580.26,Z 214.708,A -85,B 0,C 180,E1 -1779.44,E2 -1779.44} C_VEL
LIN {X 0,Y 580.24,Z 214.707,A -85,B 0,C 180,E1 -1781.647,E2 -1781.647} C_VEL
LIN {X 0,Y 580.263,Z 214.697,A -85,B 0,C 180,E1 -1784.549,E2 -1784.549} C_VEL
LIN {X 0,Y 580.244,Z 214.7,A -85,B 0,C 180,E1 -1786.698,E2 -1786.698} C_VEL
LIN {X 0,Y 580.263,Z 214.698,A -85,B 0,C 180,E1 -1788.829,E2 -1788.829} C_VEL
LIN {X 0,Y 580.299,Z 214.699,A -85,B 0,C 180,E1 -1791.646,E2 -1791.646} C_VEL
LIN {X 0,Y 580.302,Z 214.694,A -85,B 0,C 180,E1 -1794.443,E2 -1794.443} C_VEL
LIN {X 0,Y 580.331,Z 214.696,A -85,B 0,C 180,E1 -1797.92,E2 -1797.92} C_VEL
LIN {X 0,Y 580.355,Z 214.689,A -85,B 0,C 180,E1 -1800.696,E2 -1800.696} C_VEL
LIN {X 0,Y 580.33,Z 214.691,A -85,B 0,C 180,E1 -1802.779,E2 -1802.779} C_VEL
LIN {X 0,Y 580.293,Z 214.691,A -85,B 0,C 180,E1 -1805.562,E2 -1805.562} C_VEL
LIN {X 0,Y 580.258,Z 214.698,A -85,B 0,C 180,E1 -1807.658,E2 -1807.658} C_VEL
LIN {X 0,Y 580.274,Z 214.707,A -85,B 0,C 180,E1 -1810.469,E2 -1810.469} C_VEL
LIN {X 0,Y 580.294,Z 214.705,A -85,B 0,C 180,E1 -1812.594,E2 -1812.594} C_VEL
LIN {X 0,Y 580.285,Z 214.693,A -85,B 0,C 180,E1 -1815.455,E2 -1815.455} C_VEL
LIN {X 0,Y 580.265,Z 214.697,A -85,B 0,C 180,E1 -1817.627,E2 -1817.627} C_VEL
LIN {X 0,Y 580.281,Z 214.696,A -85,B 0,C 180,E1 -1819.825,E2 -1819.825} C_VEL
LIN {X 0,Y 580.257,Z 214.699,A -85,B 0,C 180,E1 -1822.055,E2 -1822.055} C_VEL
LIN {X 0,Y 580.287,Z 214.704,A -85,B 0,C 180,E1 -1825.082,E2 -1825.082} C_VEL
LIN {X 0,Y 580.252,Z 214.7,A -85,B 0,C 180,E1 -1827.85,E2 -1827.85} C_VEL
LIN {X 0,Y 580.276,Z 214.699,A -85,B 0,C 180,E1 -1830.693,E2 -1830.693} C_VEL
LIN {X 0,Y 580.287,Z 214.706,A -85,B 0,C 180,E1 -1833.313,E2 -1833.313} C_VEL
LIN {X 0,Y 580.237,Z 214.705,A -85,B 0,C 180,E1 -1835.755,E2 -1835.755} C_VEL
LIN {X 0,Y 580.29,Z 214.695,A -85,B 0,C 180,E1 -1838.148,E2 -1838.148} C_VEL
LIN {X 0,Y 580.3,Z 214.695,A -85,B 0,C 180,E1 -1840.845,E2 -1840.845} C_VEL
LIN {X 0,Y 580.245,Z 214.711,A -85,B 0,C 180,E1 -1843.662,E2 -1843.662} C_VEL
LIN {X 0,Y 580.243,Z 214.7,A -85,B 0,C 180,E1 -1846.614,E2 -1846.614} C_VEL
LIN {X 0,Y 580.287,Z 214.697,A -85,B 0,C 180,E1 -1849.155,E2 -1849.155} C_VEL
LIN {X 0,Y 580.295,Z 214.705,A -85,B 0,C 180,E1 -1851.928,E2 -1851.928} C_VEL
LIN {X 0,Y 580.238,Z 214.704,A -85,B 0,C 180,E1 -1854.451,E2 -1854.451} C_VEL
LIN {X 0,Y 580.293,Z 214.694,A -85,B 0,C 180,E1 -1856.975,E2 -1856.975} C_VEL
LIN {X 0,Y 580.289,Z 214.696,A -85,B 0,C 180,E1 -1859.424,E2 -1859.424} C_VEL
LIN {X 0,Y 580.295,Z 214.705,A -85,B 0,C 180,E1 -1862.143,E2 -1862.143} C_VEL
LIN {X 0,Y 580.295,Z 214.698,A -85,B 0,C 180,E1 -1864.919,E2 -1864.919} C_VEL
LIN {X 0,Y 580.317,Z 214.898,A -85,B 0,C 180,E1 -1867.808,E2 -1867.808} C_VEL
LIN {X 0,Y 580.805,Z 219.454,A -85,B 0,C 180,E1 -1868.547,E2 -1868.547} C_VEL
LIN {X 0,Y 580.628,Z 238.641,A -85,B 0,C 180,E1 -1871.474,E2 -1871.474} C_VEL
LIN {X 0,Y 580.475,Z 256.74,A -85,B 0,C 180,E1 -1874.192,E2 -1874.192} C_VEL
LIN {X 0,Y 580.386,Z 271.273,A -85,B 0,C 180,E1 -1876.319,E2 -1876.319} C_VEL
LIN {X 0,Y 580.98,Z 276.47,A -85,B 0,C 180,E1 -1876.422,E2 -1876.422} C_VEL
LIN {X 0,Y 580.808,Z 378.921,A -85,B 0,C 180,E1 -1877.708,E2 -1877.708} C_VEL
LIN {X 0,Y 580.744,Z 392.202,A -85,B 0,C 180,E1 -1878.017,E2 -1878.017} C_VEL
LIN {X 0,Y 580.643,Z 405.482,A -85,B 0,C 180,E1 -1878.48,E2 -1878.48} C_VEL
LIN {X 0,Y 580.564,Z 416.619,A -85,B 0,C 180,E1 -1879.008,E2 -1879.008} C_VEL
LIN {X 0,Y 580.418,Z 428.194,A -85,B 0,C 180,E1 -1879.711,E2 -1879.711} C_VEL
LIN {X 0,Y 580.343,Z 438.594,A -85,B 0,C 180,E1 -1880.502,E2 -1880.502} C_VEL
LIN {X 0,Y 580.263,Z 447.056,A -85,B 0,C 180,E1 -1881.292,E2 -1881.292} C_VEL
LIN {X 0,Y 580.223,Z 454.956,A -85,B 0,C 180,E1 -1882.168,E2 -1882.168} C_VEL
LIN {X 0,Y 580.157,Z 462.637,A -85,B 0,C 180,E1 -1883.22,E2 -1883.22} C_VEL
LIN {X 0,Y 580.139,Z 469.677,A -85,B 0,C 180,E1 -1884.438,E2 -1884.438} C_VEL
LIN {X 0,Y 580.108,Z 474.37,A -85,B 0,C 180,E1 -1885.483,E2 -1885.483} C_VEL
LIN {X 0,Y 580.123,Z 477.955,A -85,B 0,C 180,E1 -1886.527,E2 -1886.527} C_VEL
LIN {X 0,Y 580.043,Z 479.807,A -85,B 0,C 180,E1 -1887.222,E2 -1887.222} C_VEL
LIN {X 0,Y 580.038,Z 481.198,A -85,B 0,C 180,E1 -1887.916,E2 -1887.916} C_VEL
LIN {X 0,Y 580.04,Z 482.784,A -85,B 0,C 180,E1 -1889.305,E2 -1889.305} C_VEL
LIN {X 0,Y 580.037,Z 483,A -85,B 0,C 180,E1 -1889.999,E2 -1889.999} C_VEL
LIN {X 0,Y 580.046,Z 482.187,A -85,B 0,C 180,E1 -1891.388,E2 -1891.388} C_VEL
LIN {X 0,Y 580.038,Z 481.201,A -85,B 0,C 180,E1 -1892.083,E2 -1892.083} C_VEL
LIN {X 0,Y 580.043,Z 479.811,A -85,B 0,C 180,E1 -1892.777,E2 -1892.777} C_VEL
LIN {X 0,Y 580.109,Z 476.898,A -85,B 0,C 180,E1 -1893.82,E2 -1893.82} C_VEL
LIN {X 0,Y 580.053,Z 472.952,A -85,B 0,C 180,E1 -1894.865,E2 -1894.865} C_VEL
LIN {X 0,Y 580.14,Z 466.88,A -85,B 0,C 180,E1 -1896.084,E2 -1896.084} C_VEL
LIN {X 0,Y 580.185,Z 460.242,A -85,B 0,C 180,E1 -1897.132,E2 -1897.132} C_VEL
LIN {X 0,Y 580.246,Z 451.996,A -85,B 0,C 180,E1 -1898.181,E2 -1898.181} C_VEL
LIN {X 0,Y 580.333,Z 441.609,A -85,B 0,C 180,E1 -1899.233,E2 -1899.233} C_VEL
LIN {X 0,Y 580.434,Z 430.756,A -85,B 0,C 180,E1 -1900.111,E2 -1900.111} C_VEL
LIN {X 0,Y 580.537,Z 419.795,A -85,B 0,C 180,E1 -1900.815,E2 -1900.815} C_VEL
LIN {X 0,Y 580.663,Z 407.56,A -85,B 0,C 180,E1 -1901.429,E2 -1901.429} C_VEL
LIN {X 0,Y 580.732,Z 395.891,A -85,B 0,C 180,E1 -1901.872,E2 -1901.872} C_VEL
LIN {X 0,Y 580.786,Z 383.541,A -85,B 0,C 180,E1 -1902.203,E2 -1902.203} C_VEL
LIN {X 0,Y 580.832,Z 367.788,A -85,B 0,C 180,E1 -1902.446,E2 -1902.446} C_VEL
LIN {X 0,Y 580.903,Z 274.776,A -85,B 0,C 180,E1 -1903.6,E2 -1903.6} C_VEL
LIN {X 0,Y 580.386,Z 271.294,A -85,B 0,C 180,E1 -1903.68,E2 -1903.68} C_VEL
LIN {X 0,Y 580.501,Z 253.128,A -85,B 0,C 180,E1 -1906.348,E2 -1906.348} C_VEL
LIN {X 0,Y 580.647,Z 235.029,A -85,B 0,C 180,E1 -1909.074,E2 -1909.074} C_VEL
LIN {X 0,Y 580.817,Z 218.123,A -85,B 0,C 180,E1 -1911.656,E2 -1911.656} C_VEL
LIN {X 0,Y 580.306,Z 214.769,A -85,B 0,C 180,E1 -1912.238,E2 -1912.238} C_VEL
LIN {X 0,Y 580.292,Z 214.698,A -85,B 0,C 180,E1 -1915.08,E2 -1915.08} C_VEL
LIN {X 0,Y 580.296,Z 214.705,A -85,B 0,C 180,E1 -1917.857,E2 -1917.857} C_VEL
LIN {X 0,Y 580.282,Z 214.697,A -85,B 0,C 180,E1 -1920.693,E2 -1920.693} C_VEL
LIN {X 0,Y 580.303,Z 214.695,A -85,B 0,C 180,E1 -1923.315,E2 -1923.315} C_VEL
LIN {X 0,Y 580.243,Z 214.707,A -85,B 0,C 180,E1 -1925.755,E2 -1925.755} C_VEL
LIN {X 0,Y 580.285,Z 214.706,A -85,B 0,C 180,E1 -1928.145,E2 -1928.145} C_VEL
LIN {X 0,Y 580.293,Z 214.695,A -85,B 0,C 180,E1 -1930.843,E2 -1930.843} C_VEL
LIN {X 0,Y 580.238,Z 214.703,A -85,B 0,C 180,E1 -1933.66,E2 -1933.66} C_VEL
LIN {X 0,Y 580.264,Z 214.704,A -85,B 0,C 180,E1 -1936.609,E2 -1936.609} C_VEL
LIN {X 0,Y 580.292,Z 214.695,A -85,B 0,C 180,E1 -1939.155,E2 -1939.155} C_VEL
LIN {X 0,Y 580.284,Z 214.697,A -85,B 0,C 180,E1 -1941.926,E2 -1941.926} C_VEL
LIN {X 0,Y 580.245,Z 214.71,A -85,B 0,C 180,E1 -1944.451,E2 -1944.451} C_VEL
LIN {X 0,Y 580.284,Z 214.7,A -85,B 0,C 180,E1 -1946.973,E2 -1946.973} C_VEL
LIN {X 0,Y 580.277,Z 214.697,A -85,B 0,C 180,E1 -1949.422,E2 -1949.422} C_VEL
LIN {X 0,Y 580.241,Z 214.702,A -85,B 0,C 180,E1 -1952.15,E2 -1952.15} C_VEL
LIN {X 0,Y 580.278,Z 214.706,A -85,B 0,C 180,E1 -1954.917,E2 -1954.917} C_VEL
LIN {X 0,Y 580.247,Z 214.7,A -85,B 0,C 180,E1 -1957.945,E2 -1957.945} C_VEL
LIN {X 0,Y 580.293,Z 214.703,A -85,B 0,C 180,E1 -1960.848,E2 -1960.848} C_VEL
LIN {X 0,Y 580.243,Z 214.702,A -85,B 0,C 180,E1 -1963.823,E2 -1963.823} C_VEL
LIN {X 0,Y 580.271,Z 214.697,A -85,B 0,C 180,E1 -1965.98,E2 -1965.98} C_VEL
LIN {X 0,Y 580.3,Z 214.697,A -85,B 0,C 180,E1 -1968.825,E2 -1968.825} C_VEL
LIN {X 0,Y 580.278,Z 214.701,A -85,B 0,C 180,E1 -1971.641,E2 -1971.641} C_VEL
LIN {X 0,Y 580.244,Z 214.705,A -85,B 0,C 180,E1 -1973.74,E2 -1973.74} C_VEL
LIN {X 0,Y 580.225,Z 214.706,A -85,B 0,C 180,E1 -1975.83,E2 -1975.83} C_VEL
LIN {X 0,Y 580.301,Z 214.697,A -85,B 0,C 180,E1 -1977.916,E2 -1977.916} C_VEL
LIN {X 0,Y 580.314,Z 214.695,A -85,B 0,C 180,E1 -1979.998,E2 -1979.998} C_VEL
LIN {X 0,Y 580.284,Z 214.696,A -85,B 0,C 180,E1 -1982.774,E2 -1982.774} C_VEL
LIN {X 0,Y 580.285,Z 214.703,A -85,B 0,C 180,E1 -1985.558,E2 -1985.558} C_VEL
LIN {X 0,Y 580.278,Z 214.698,A -85,B 0,C 180,E1 -1988.354,E2 -1988.354} C_VEL
LIN {X 0,Y 580.252,Z 214.701,A -85,B 0,C 180,E1 -1991.171,E2 -1991.171} C_VEL
LIN {X 0,Y 580.293,Z 214.705,A -85,B 0,C 180,E1 -1994.015,E2 -1994.015} C_VEL
LIN {X 0,Y 580.249,Z 214.7,A -85,B 0,C 180,E1 -1996.896,E2 -1996.896} C_VEL
LIN {X 0,Y 580.262,Z 214.704,A -85,B 0,C 180,E1 -1999.821,E2 -1999.821} C_VEL
LIN {X 0,Y 580.267,Z 214.698,A -85,B 0,C 180,E1 -2001.275,E2 -2001.275} C_VEL
LIN {X 0,Y 579.554,Z 214.794,A -85,B 0,C 180,E1 -2001.854,E2 -2001.854} C_VEL
LIN {X 0,Y 576.673,Z 215.148,A -85,B 0,C 180,E1 -2002.794,E2 -2002.794} C_VEL
LIN {X 0,Y 574.283,Z 215.445,A -85,B 0,C 180,E1 -2003.55,E2 -2003.55} C_VEL
LIN {X 0,Y 573.286,Z 215.576,A -85,B 0,C 180,E1 -2004.134,E2 -2004.134} C_VEL
LIN {X 0,Y 573.219,Z 215.579,A -85,B 0,C 180,E1 -2004.332,E2 -2004.332} C_VEL
LIN {X 0,Y 573.177,Z 215.583,A -85,B 0,C 180,E1 -2006.976,E2 -2006.976} C_VEL
LIN {X 0,Y 573.216,Z 215.576,A -85,B 0,C 180,E1 -2009.485,E2 -2009.485} C_VEL
LIN {X 0,Y 573.229,Z 215.583,A -85,B 0,C 180,E1 -2012.643,E2 -2012.643} C_VEL
LIN {X 0,Y 573.239,Z 215.575,A -85,B 0,C 180,E1 -2015.181,E2 -2015.181} C_VEL
LIN {X 0,Y 573.207,Z 215.578,A -85,B 0,C 180,E1 -2017.805,E2 -2017.805} C_VEL
LIN {X 0,Y 573.24,Z 215.582,A -85,B 0,C 180,E1 -2020.526,E2 -2020.526} C_VEL
LIN {X 0,Y 573.225,Z 215.577,A -85,B 0,C 180,E1 -2023.668,E2 -2023.668} C_VEL
LIN {X 0,Y 573.282,Z 215.71,A -85,B 0,C 180,E1 -2026.37,E2 -2026.37} C_VEL
LIN {X 0,Y 573.683,Z 219.537,A -85,B 0,C 180,E1 -2027.032,E2 -2027.032} C_VEL
LIN {X 0,Y 573.452,Z 237.072,A -85,B 0,C 180,E1 -2029.954,E2 -2029.954} C_VEL
LIN {X 0,Y 573.318,Z 252.731,A -85,B 0,C 180,E1 -2032.545,E2 -2032.545} C_VEL
LIN {X 0,Y 573.332,Z 256.931,A -85,B 0,C 180,E1 -2033.198,E2 -2033.198} C_VEL
LIN {X 0,Y 574.006,Z 261.503,A -85,B 0,C 180,E1 -2033.3,E2 -2033.3} C_VEL
LIN {X 0,Y 573.881,Z 364.099,A -85,B 0,C 180,E1 -2034.605,E2 -2034.605} C_VEL
LIN {X 0,Y 573.816,Z 376.791,A -85,B 0,C 180,E1 -2034.903,E2 -2034.903} C_VEL
LIN {X 0,Y 573.728,Z 389.393,A -85,B 0,C 180,E1 -2035.34,E2 -2035.34} C_VEL
LIN {X 0,Y 573.586,Z 401.327,A -85,B 0,C 180,E1 -2035.901,E2 -2035.901} C_VEL
LIN {X 0,Y 573.413,Z 413.255,A -85,B 0,C 180,E1 -2036.633,E2 -2036.633} C_VEL
LIN {X 0,Y 573.334,Z 424.17,A -85,B 0,C 180,E1 -2037.478,E2 -2037.478} C_VEL
LIN {X 0,Y 573.219,Z 433.62,A -85,B 0,C 180,E1 -2038.391,E2 -2038.391} C_VEL
LIN {X 0,Y 573.123,Z 442.233,A -85,B 0,C 180,E1 -2039.41,E2 -2039.41} C_VEL
LIN {X 0,Y 573.071,Z 449.87,A -85,B 0,C 180,E1 -2040.535,E2 -2040.535} C_VEL
LIN {X 0,Y 573.026,Z 456.268,A -85,B 0,C 180,E1 -2041.746,E2 -2041.746} C_VEL
LIN {X 0,Y 572.988,Z 461.334,A -85,B 0,C 180,E1 -2043.012,E2 -2043.012} C_VEL
LIN {X 0,Y 572.996,Z 463.716,A -85,B 0,C 180,E1 -2043.798,E2 -2043.798} C_VEL
LIN {X 0,Y 572.949,Z 466.587,A -85,B 0,C 180,E1 -2045.181,E2 -2045.181} C_VEL
LIN {X 0,Y 572.944,Z 467.638,A -85,B 0,C 180,E1 -2046.123,E2 -2046.123} C_VEL
LIN {X 0,Y 572.945,Z 467.977,A -85,B 0,C 180,E1 -2046.913,E2 -2046.913} C_VEL
LIN {X 0,Y 572.936,Z 467.849,A -85,B 0,C 180,E1 -2047.651,E2 -2047.651} C_VEL
LIN {X 0,Y 572.952,Z 466.796,A -85,B 0,C 180,E1 -2048.775,E2 -2048.775} C_VEL
LIN {X 0,Y 572.973,Z 463.726,A -85,B 0,C 180,E1 -2050.288,E2 -2050.288} C_VEL
LIN {X 0,Y 573.005,Z 460.186,A -85,B 0,C 180,E1 -2051.405,E2 -2051.405} C_VEL
LIN {X 0,Y 573.034,Z 455.489,A -85,B 0,C 180,E1 -2052.514,E2 -2052.514} C_VEL
LIN {X 0,Y 573.071,Z 449.485,A -85,B 0,C 180,E1 -2053.617,E2 -2053.617} C_VEL
LIN {X 0,Y 573.159,Z 441.958,A -85,B 0,C 180,E1 -2054.715,E2 -2054.715} C_VEL
LIN {X 0,Y 573.236,Z 433.694,A -85,B 0,C 180,E1 -2055.691,E2 -2055.691} C_VEL
LIN {X 0,Y 573.332,Z 424.038,A -85,B 0,C 180,E1 -2056.623,E2 -2056.623} C_VEL
LIN {X 0,Y 573.43,Z 413.549,A -85,B 0,C 180,E1 -2057.436,E2 -2057.436} C_VEL
LIN {X 0,Y 573.552,Z 401.631,A -85,B 0,C 180,E1 -2058.172,E2 -2058.172} C_VEL
LIN {X 0,Y 573.69,Z 389.612,A -85,B 0,C 180,E1 -2058.742,E2 -2058.742} C_VEL
LIN {X 0,Y 573.773,Z 376.722,A -85,B 0,C 180,E1 -2059.19,E2 -2059.19} C_VEL
LIN {X 0,Y 573.879,Z 364.211,A -85,B 0,C 180,E1 -2059.482,E2 -2059.482} C_VEL
LIN {X 0,Y 573.872,Z 260.478,A -85,B 0,C 180,E1 -2060.807,E2 -2060.807} C_VEL
LIN {X 0,Y 573.344,Z 257.194,A -85,B 0,C 180,E1 -2060.876,E2 -2060.876} C_VEL
LIN {X 0,Y 573.31,Z 254.912,A -85,B 0,C 180,E1 -2061.186,E2 -2061.186} C_VEL
LIN {X 0,Y 573.487,Z 237.753,A -85,B 0,C 180,E1 -2064.022,E2 -2064.022} C_VEL
LIN {X 0,Y 573.648,Z 219.908,A -85,B 0,C 180,E1 -2067.016,E2 -2067.016} C_VEL
LIN {X 0,Y 573.262,Z 215.64,A -85,B 0,C 180,E1 -2067.805,E2 -2067.805} C_VEL
LIN {X 0,Y 573.27,Z 215.572,A -85,B 0,C 180,E1 -2070.001,E2 -2070.001} C_VEL
LIN {X 0,Y 573.272,Z 215.573,A -85,B 0,C 180,E1 -2072.811,E2 -2072.811} C_VEL
LIN {X 0,Y 573.266,Z 215.578,A -85,B 0,C 180,E1 -2075.629,E2 -2075.629} C_VEL
LIN {X 0,Y 573.245,Z 215.573,A -85,B 0,C 180,E1 -2078.461,E2 -2078.461} C_VEL
LIN {X 0,Y 573.232,Z 215.579,A -85,B 0,C 180,E1 -2081.313,E2 -2081.313} C_VEL
LIN {X 0,Y 573.221,Z 215.579,A -85,B 0,C 180,E1 -2084.195,E2 -2084.195} C_VEL
LIN {X 0,Y 573.222,Z 215.576,A -85,B 0,C 180,E1 -2087.113,E2 -2087.113} C_VEL
LIN {X 0,Y 573.213,Z 215.585,A -85,B 0,C 180,E1 -2090.079,E2 -2090.079} C_VEL
LIN {X 0,Y 573.199,Z 215.578,A -85,B 0,C 180,E1 -2093.101,E2 -2093.101} C_VEL
LIN {X 0,Y 573.211,Z 215.577,A -85,B 0,C 180,E1 -2095.413,E2 -2095.413} C_VEL
LIN {X 0,Y 573.191,Z 215.582,A -85,B 0,C 180,E1 -2098.567,E2 -2098.567} C_VEL
LIN {X 0,Y 573.194,Z 215.58,A -85,B 0,C 180,E1 -2100.996,E2 -2100.996} C_VEL
LIN {X 0,Y 573.21,Z 215.577,A -85,B 0,C 180,E1 -2103.523,E2 -2103.523} C_VEL
LIN {X 0,Y 573.157,Z 215.586,A -85,B 0,C 180,E1 -2106.056,E2 -2106.056} C_VEL
LIN {X 0,Y 573.201,Z 215.586,A -85,B 0,C 180,E1 -2108.705,E2 -2108.705} C_VEL
LIN {X 0,Y 573.173,Z 215.58,A -85,B 0,C 180,E1 -2111.462,E2 -2111.462} C_VEL
LIN {X 0,Y 573.19,Z 215.582,A -85,B 0,C 180,E1 -2114.338,E2 -2114.338} C_VEL
LIN {X 0,Y 573.194,Z 215.581,A -85,B 0,C 180,E1 -2117.364,E2 -2117.364} C_VEL
LIN {X 0,Y 573.208,Z 215.578,A -85,B 0,C 180,E1 -2120.394,E2 -2120.394} C_VEL
LIN {X 0,Y 573.231,Z 215.583,A -85,B 0,C 180,E1 -2123.08,E2 -2123.08} C_VEL
LIN {X 0,Y 573.234,Z 215.576,A -85,B 0,C 180,E1 -2125.673,E2 -2125.673} C_VEL
LIN {X 0,Y 573.206,Z 215.576,A -85,B 0,C 180,E1 -2128.186,E2 -2128.186} C_VEL
LIN {X 0,Y 573.217,Z 215.575,A -85,B 0,C 180,E1 -2130.635,E2 -2130.635} C_VEL
LIN {X 0,Y 573.18,Z 215.587,A -85,B 0,C 180,E1 -2133.519,E2 -2133.519} C_VEL
LIN {X 0,Y 573.195,Z 215.579,A -85,B 0,C 180,E1 -2136.136,E2 -2136.136} C_VEL
LIN {X 0,Y 573.239,Z 215.578,A -85,B 0,C 180,E1 -2139.176,E2 -2139.176} C_VEL
LIN {X 0,Y 573.197,Z 215.584,A -85,B 0,C 180,E1 -2141.414,E2 -2141.414} C_VEL
LIN {X 0,Y 573.204,Z 215.577,A -85,B 0,C 180,E1 -2144.354,E2 -2144.354} C_VEL
LIN {X 0,Y 573.205,Z 215.578,A -85,B 0,C 180,E1 -2146.532,E2 -2146.532} C_VEL
LIN {X 0,Y 573.236,Z 215.577,A -85,B 0,C 180,E1 -2149.406,E2 -2149.406} C_VEL
LIN {X 0,Y 573.219,Z 215.578,A -85,B 0,C 180,E1 -2152.252,E2 -2152.252} C_VEL
LIN {X 0,Y 573.274,Z 215.565,A -85,B 0,C 180,E1 -2155.08,E2 -2155.08} C_VEL
LIN {X 0,Y 573.301,Z 215.571,A -85,B 0,C 180,E1 -2157.895,E2 -2157.895} C_VEL
LIN {X 0,Y 573.326,Z 215.565,A -85,B 0,C 180,E1 -2160.705,E2 -2160.705} C_VEL
LIN {X 0,Y 573.294,Z 215.567,A -85,B 0,C 180,E1 -2162.813,E2 -2162.813} C_VEL
LIN {X 0,Y 573.263,Z 215.567,A -85,B 0,C 180,E1 -2165.631,E2 -2165.631} C_VEL
LIN {X 0,Y 573.216,Z 215.576,A -85,B 0,C 180,E1 -2167.753,E2 -2167.753} C_VEL
LIN {X 0,Y 573.248,Z 215.582,A -85,B 0,C 180,E1 -2170.599,E2 -2170.599} C_VEL
LIN {X 0,Y 573.215,Z 215.575,A -85,B 0,C 180,E1 -2173.473,E2 -2173.473} C_VEL
LIN {X 0,Y 573.238,Z 215.575,A -85,B 0,C 180,E1 -2176.381,E2 -2176.381} C_VEL
LIN {X 0,Y 573.273,Z 215.572,A -85,B 0,C 180,E1 -2179.332,E2 -2179.332} C_VEL
LIN {X 0,Y 573.228,Z 215.575,A -85,B 0,C 180,E1 -2181.582,E2 -2181.582} C_VEL
LIN {X 0,Y 573.203,Z 215.575,A -85,B 0,C 180,E1 -2183.868,E2 -2183.868} C_VEL
LIN {X 0,Y 573.238,Z 215.575,A -85,B 0,C 180,E1 -2186.492,E2 -2186.492} C_VEL
LIN {X 0,Y 573.228,Z 215.578,A -85,B 0,C 180,E1 -2189.484,E2 -2189.484} C_VEL
LIN {X 0,Y 573.245,Z 215.571,A -85,B 0,C 180,E1 -2192.227,E2 -2192.227} C_VEL
LIN {X 0,Y 573.229,Z 215.577,A -85,B 0,C 180,E1 -2194.77,E2 -2194.77} C_VEL
LIN {X 0,Y 573.236,Z 215.577,A -85,B 0,C 180,E1 -2197.809,E2 -2197.809} C_VEL
LIN {X 0,Y 573.254,Z 215.571,A -85,B 0,C 180,E1 -2200.526,E2 -2200.526} C_VEL
LIN {X 0,Y 573.208,Z 215.583,A -85,B 0,C 180,E1 -2203.363,E2 -2203.363} C_VEL
LIN {X 0,Y 573.214,Z 215.577,A -85,B 0,C 180,E1 -2206.336,E2 -2206.336} C_VEL
LIN {X 0,Y 573.215,Z 215.577,A -85,B 0,C 180,E1 -2208.541,E2 -2208.541} C_VEL
LIN {X 0,Y 573.243,Z 215.575,A -85,B 0,C 180,E1 -2211.298,E2 -2211.298} C_VEL
LIN {X 0,Y 573.195,Z 215.588,A -85,B 0,C 180,E1 -2214.022,E2 -2214.022} C_VEL
LIN {X 0,Y 573.26,Z 215.573,A -85,B 0,C 180,E1 -2216.517,E2 -2216.517} C_VEL
LIN {X 0,Y 573.228,Z 215.575,A -85,B 0,C 180,E1 -2219.119,E2 -2219.119} C_VEL
LIN {X 0,Y 573.249,Z 215.58,A -85,B 0,C 180,E1 -2221.973,E2 -2221.973} C_VEL
LIN {X 0,Y 573.246,Z 215.58,A -85,B 0,C 180,E1 -2224.589,E2 -2224.589} C_VEL
LIN {X 0,Y 573.291,Z 215.741,A -85,B 0,C 180,E1 -2227.664,E2 -2227.664} C_VEL
LIN {X 0,Y 573.856,Z 220.474,A -85,B 0,C 180,E1 -2228.444,E2 -2228.444} C_VEL
LIN {X 0,Y 573.666,Z 239.847,A -85,B 0,C 180,E1 -2231.426,E2 -2231.426} C_VEL
LIN {X 0,Y 573.431,Z 259.153,A -85,B 0,C 180,E1 -2234.357,E2 -2234.357} C_VEL
